// TwinCAT 3 PLC project PunchingMachine
// ProgramVersion: 3.1.4026.20
// libraries:
//   RMTH TC3 Library, * (RMTH GmbH)
//   Tc2_Drive, * (Beckhoff Automation GmbH)
//   Tc2_EtherCAT, * (Beckhoff Automation GmbH)
//   Tc2_MC2, * (Beckhoff Automation GmbH)
//   Tc2_MC2_Drive, * (Beckhoff Automation GmbH)
//   Tc2_NC, * (Beckhoff Automation GmbH)
//   Tc2_NCI, * (Beckhoff Automation GmbH)
//   Tc2_Standard, * (Beckhoff Automation GmbH)
//   Tc2_System, * (Beckhoff Automation GmbH)
//   Tc2_Utilities, * (Beckhoff Automation GmbH)
//   Tc3_EventLogger, * (Beckhoff Automation GmbH)
//   Tc3_Module, * (Beckhoff Automation GmbH)
//   BASIC,3.3.3.0,OSCAT
// project tree:
//   BaseComponents/AxisDriver/Enumeration/ E_GearMode.TcDUT, E_JogDirection.TcDUT, E_MotionCommand.TcDUT
//   BaseComponents/AxisDriver/ FB_AxisDriver.TcPOU
//   BaseComponents/AxisDriver/Interfaces/ ITFMotionComponent.TcIO
//   BaseComponents/AxisDriver/Structures/AdditionalAxisIO/ ST_AxisIn.TcDUT, ST_AxisIO.TcDUT, ST_AxisOut.TcDUT, ST_AxisVirtualIO.TcDUT
//   BaseComponents/AxisDriver/Structures/ ST_AxisDriverParameter.TcDUT, ST_AxisGearInParameter.TcDUT, ST_AxisGearOutParameter.TcDUT, ST_AxisGeneralParameter.TcDUT, ST_AxisHaltParameter.TcDUT, ST_AxisHomingParameter.TcDUT, ST_AxisJogAccParameter.TcDUT, ST_AxisJogParameter.TcDUT, ST_AxisMoveAbsParameter.TcDUT, ST_AxisMoveAddParameter.TcDUT, ST_AxisMoveModParameter.TcDUT, ST_AxisMoveParameter.TcDUT, ST_AxisMoveRelParameter.TcDUT, ST_AxisMoveVelParameter.TcDUT, ST_AxisSetPosParameter.TcDUT, ST_AxisStopParameter.TcDUT
//   BaseComponents/AxisDriver/Utilities/ FB_AxisDistanceTrigger.TcPOU, FB_LimitSwitchRefSim.TcPOU, F_LRealToString.TcPOU, F_LRealToStringEx.TcPOU, F_SpeedReached.TcPOU, F_SpeedWindowReached.TcPOU, F_TargetReached.TcPOU, F_TargetReachedOrHigher.TcPOU, F_TargetReachedOrLower.TcPOU, F_TargetWindowReached.TcPOU, F_TargetWindowReachedAxisRef.TcPOU
//   BaseComponents/CylinderDriver/Enumeration/ E_CylinderPosition.TcDUT
//   BaseComponents/CylinderDriver/ FB_CylinderDriver.TcPOU
//   BaseComponents/CylinderDriver/Interfaces/ ITF_Cylinder.TcIO
//   BaseComponents/CylinderDriver/Structures/ ST_CylinderDriverIn.TcDUT, ST_CylinderDriverIO.TcDUT, ST_CylinderDriverOut.TcDUT
//   BaseComponents/DigitalInput/ FB_DigitalInput.TcPOU
//   BaseComponents/DigitalInput/Structures/ ST_DigitalInputIn.TcDUT, ST_DigitalInputIO.TcDUT
//   BaseComponents/DigitalOutput/ FB_DigitalOutput.TcPOU
//   BaseComponents/DigitalOutput/Structures/ ST_DigitalOutputIO.TcDUT, ST_DigitalOutputOUT.TcDUT
//   BaseComponents/EtherCAT/Enumerations/ E_EtherCatSlaveState.TcDUT, E_EtherCATState.TcDUT
//   BaseComponents/EtherCAT/ FB_EtherCatBox.TcPOU, FB_EtherCATBus.TcPOU
//   BaseComponents/EtherCAT/Structures/ ST_EtherCatBoxIO.TcDUT, ST_EtherCatIO.TcDUT
//   BaseComponents/EventLog/Enumerations/ E_BoolFilter.TcDUT, E_FilterActive.TcDUT, E_Priority.TcDUT
//   BaseComponents/EventLog/ E_Event.TcDUT, FB_EventLog.TcPOU
//   BaseComponents/EventLog/Structures/ ST_Event.TcDUT, ST_EventFilter.TcDUT
//   BaseComponents/SafetyLockDriver/ FB_SafetyLock.TcPOU
//   BaseComponents/SafetyLockDriver/Structures/ ST_SafetyLockIn.TcDUT, ST_SafetyLockIO.TcDUT, ST_SafetyLockOut.TcDUT
//   BaseComponents/Safety/ FB_Safety.TcPOU
//   BaseComponents/Safety/Structures/ ST_SafetyIn.TcDUT, ST_SafetyIO.TcDUT, ST_SafetyOut.TcDUT
//   BaseComponents/Supervision/CheckFunctions/ CheckBounds.TcPOU, CheckDivDInt.TcPOU, CheckDivLInt.TcPOU, CheckDivLReal.TcPOU, CheckDivReal.TcPOU, CheckPointer.TcPOU, CheckRangeSigned.TcPOU, CheckRangeUnsigned.TcPOU
//   BaseComponents/Supervision/Enumeration/ E_CodeError.TcDUT
//   BaseComponents/Supervision/ FB_Supervision.TcPOU, GVL_Supervision.TcGVL
//   Components/ E_ComponentType.TcDUT
//   Components/MatAndToolHandling/Enumerations/ E_MatAndToolHandlingCmd.TcDUT
//   Components/MatAndToolHandling/ FB_MatAndToolHandling.TcPOU
//   Components/Mat/Enumerations/ E_CoordinatesSortState.TcTLEO, E_Geometry.TcDUT, E_ElementOrigin.TcDUT
//   Components/Mat/ FB_Mat.TcPOU
//   Components/Mat/Structures/ ST_Element.TcDUT, ST_Mat.TcDUT, ST_MatRun.TcDUT, ST_Tool.TcDUT, ST_ToolHolder.TcDUT, ST_Coordinate.TcDUT
//   Components/PunchEngine/Enumerations/ E_PunchEngineCmd.TcDUT
//   Components/PunchEngine/ FB_PunchEngine.TcPOU
//   / IOTask.TcTTO, NcTask.TcTTO, PlcTask.TcTTO, VisuTask.TcTTO
//   Machine/Components/ E_Axis.TcDUT, E_DigitalOutput.TcDUT, E_Cylinder.TcDUT, COMP_CONST.TcGVL, COMP.TcGVL
//   Machine/Enumerations/ E_JobState.TcDUT, E_MachineArea.TcDUT, E_OperationMode.TcDUT, E_RunTodo.TcDUT
//   Machine/ GVL.TcGVL, GVL_CONST.TcGVL, P_Machine.TcPOU
//   Machine/Structures/ ST_MachineConfig.TcDUT, ST_PunchJob.TcDUT
//   Utilities/Component/Enumerations/ E_ComponentState.TcDUT
//   Utilities/Component/ FB_ComponentBase.TcPOU
//   Utilities/Component/Interfaces/ ITFComponent.TcIO
//   Utilities/Composition/ FB_CompositionBase.TcPOU
//   Utilities/Sequencer/Enumeration/ E_SequenceState.TcDUT
//   Utilities/Sequencer/ FB_Sequence.TcPOU
//   Utilities/TaskAllocation/Enumerations/ E_Task.TcDUT
//   Utilities/TaskAllocation/ P_Fast.TcPOU
//   Utilities/TaskAllocation/Interfaces/ ITF_TaskAllocation.TcIO
//   Visualisation/Structures/ ST_MaintCmds.TcDUT, ST_MaintParam.TcDUT, ST_PunchCmds.TcDUT, ST_PunchInfo.TcDUT, ST_MaintInfo.TcDUT, ST_PunchParam.TcDUT
//   Visualisation/ GVL_VISU.TcGVL, P_Visu.TcPOU
// real-time tasks:
//   TASK PlcTask: cycle T#10ms, priority 14, ADS port 350
//   TASK NcTask: cycle T#10ms, priority 12, ADS port 351
//   TASK IOTask: cycle T#10ms, priority 8, ADS port 354
//   TASK VisuTask: cycle T#50000us, priority 16, ADS port 353
// motion (NC):
//   TASK NC-Task 1 SAF: cycle T#2ms, priority 4, ADS port 501
//   TASK NC-Task 1 SVB: cycle T#10ms, priority 10, ADS port 511
//   AXIS x-Axis (id 4)
//     Dynamic: Acceleration=5500, Deceleration=5500, Jerk=15000
//     Velo: RefSearch=18.6430234375, RefSync=18.6430234375, SlowManual=10, FastManual=250, Fast=1864.30234375, Maximum=1864.3
//     OtherSettings: AllowMotionCmdToSlave=true
//     encoder EncType=8
//       EncPara: ScaleFactorNumerator=41.5555555555556, ScaleFactorDenominator=1048576, Offset=17493, MaxCount=#xffffffff
//         SoftEndMinControl: Enable=true
//         SoftEndMaxControl: Enable=true, Range=4070
//     drive DrvType=9
//       DrvPara: MaxCount=#xffffffff, DriveControlDWord=#x00030100
//         Analog: VeloReferenz=2050.732578125, VeloScale=1.02400649589962, ScaleFactorActTorque=0.1
//         TimeComp: TaskDelayCycles=1
//     controller CtrType=1
//       CtrPara: PriorControlFactor=1
//         Observer: BandWidth=20
//   AXIS y-Axis (id 5)
//     Dynamic: Acceleration=11000, Deceleration=11000, Jerk=30000
//     Velo: RefSearch=32.25, RefSync=32.25, SlowManual=161.25, FastManual=967.5, Fast=3225, Maximum=3225
//     OtherSettings: AllowMotionCmdToSlave=true
//     encoder EncType=8
//       EncPara: ScaleFactorNumerator=21.5, ScaleFactorDenominator=1048576, Offset=-280, Inverse=true, MaxCount=#xffffffff
//         SoftEndMinControl: Enable=true, Range=5
//         SoftEndMaxControl: Enable=true, Range=790
//     drive DrvType=9
//       DrvPara: Inverse=true, MaxCount=#xffffffff, DriveControlDWord=#x00030100
//         Analog: VeloReferenz=3547.5, VeloScale=1.02400649589962, ScaleFactorActTorque=0.1
//         TimeComp: TaskDelayCycles=1
//     controller CtrType=1
//       CtrPara: PriorControlFactor=1
//         Observer: BandWidth=20
//   AXIS PunchAxis (id 6)
//     General: UnitName=Degree, UnitFlags=#x00000004
//     Dynamic: Acceleration=10000, Deceleration=10000, Jerk=100000
//     Velo: RefSearch=11.1429969216489, RefSync=11.1429969216489, SlowManual=55.7149846082443, FastManual=900, Fast=1114.29969216489, Maximum=1114.3
//     PositionAreaControl: Enable=false
//     TargetPosControl: Enable=false
//     OtherSettings: AllowMotionCmdToSlave=true
//     encoder EncType=8
//       EncPara: ScaleFactorNumerator=20.1237295625276, ScaleFactorDenominator=1048576, Offset=-12, ToleranceWndModuloStart=1.5, MaxCount=#x000fffff
//     drive DrvType=9
//       DrvPara: MaxCount=#xffffffff, DriveControlDWord=#x00030100
//         Analog: VeloReferenz=1225.72966138138, VeloScale=1.02400649589962, ScaleFactorActTorque=0.1
//         TimeComp: TaskDelayCycles=1
//     controller CtrType=1
//       CtrPara: PriorControlFactor=1
//         PosDiffControl: Enable=false
//         Observer: BandWidth=20
// I/O:
//   DEVICE Device 2 (EtherCAT), AmsNetId 192.168.137.129.3.1
//     Term 1 (EK1100) [EK1100 EtherCAT Coupler (2A E-Bus)]
//       Term 2 (EL6910) [EL6910, TwinSAFE PLC]
//       Term 3 (EL2904) [EL2904, 4 Ch. Safety Output 24V, 0.5A, TwinSAFE]
//         modules: Module 1 (FSOES), Module 2 (DO)
//       Term 4 (EL1904) [EL1904, 4 Ch. Safety Input 24V, TwinSAFE]
//         modules: Module 1 (FSOES)
//       Term 5 (EL1904) [EL1904, 4 Ch. Safety Input 24V, TwinSAFE]
//         modules: Module 1 (FSOES)
//       Term 6 (EL1008) [EL1008 8Ch. Dig. Input 24V, 3ms]
//       Term 7 (EL1008) [EL1008 8Ch. Dig. Input 24V, 3ms]
//       Term 8 (EL2008) [EL2008 8Ch. Dig. Output 24V, 0.5A]
//       Term 13 (EL9011) [EL9011 End Terminal]
//     Drive 9 (AX5206-0000-0210) [AX5206-0000-0210 EtherCAT Drive (SoE, 2 Ch.)]
//       Term 10 (AX5805) [AX5805 (Safety Drive Option)]
//         modules: Module 1 (Safety Process Data, 2 axis), Module 2 (Standard Process Data, 2 axis)
//       Term 14 (EL9011) [EL9011 End Terminal]
//     Drive 11 (AX5112-0000-0210) [AX5112-0000-0210 EtherCAT Drive (SoE, 1 Ch.)]
//       Term 12 (AX5805) [AX5805 (Safety Drive Option)]
//         modules: Module 1 (Safety Process Data, 1 axis), Module 2 (Standard Process Data, 1 axis)
//       Term 15 (EL9011) [EL9011 End Terminal]
// variable links:
//   Device 2 (EtherCAT) <-> Device 2 (EtherCAT)/Drive 11 (AX5112-0000-0210)/Term 12 (AX5805)
//     Term 1 (EK1100)/Term 2 (EL6910)/ConnectionInputs/Message_7 TxPDO <-> Module 1 (Safety Process Data, 1 axis)/Outputs (Controlword)/FSOE
//     Term 1 (EK1100)/Term 2 (EL6910)/ConnectionOutputs/Message_7 RxPDO <-> Module 1 (Safety Process Data, 1 axis)/Inputs (Statusword)/FSOE
//   Device 2 (EtherCAT) <-> Device 2 (EtherCAT)/Drive 9 (AX5206-0000-0210)/Term 10 (AX5805)
//     Term 1 (EK1100)/Term 2 (EL6910)/ConnectionInputs/Message_6 TxPDO <-> Module 1 (Safety Process Data, 2 axis)/Outputs (Controlword)/FSOE
//     Term 1 (EK1100)/Term 2 (EL6910)/ConnectionOutputs/Message_6 RxPDO <-> Module 1 (Safety Process Data, 2 axis)/Inputs (Statusword)/FSOE
//   Device 2 (EtherCAT) <-> Device 2 (EtherCAT)/Term 1 (EK1100)/Term 3 (EL2904)
//     Term 1 (EK1100)/Term 2 (EL6910)/ConnectionInputs/Message_16 TxPDO <-> Module 1 (FSOES)/RxPDO/FSOE
//     Term 1 (EK1100)/Term 2 (EL6910)/ConnectionOutputs/Message_16 RxPDO <-> Module 1 (FSOES)/TxPDO/FSOE
//   Device 2 (EtherCAT) <-> Device 2 (EtherCAT)/Term 1 (EK1100)/Term 4 (EL1904)
//     Term 1 (EK1100)/Term 2 (EL6910)/ConnectionInputs/Message_4 TxPDO <-> Module 1 (FSOES)/RxPDO/FSOE
//     Term 1 (EK1100)/Term 2 (EL6910)/ConnectionOutputs/Message_4 RxPDO <-> Module 1 (FSOES)/TxPDO/FSOE
//   Device 2 (EtherCAT) <-> Device 2 (EtherCAT)/Term 1 (EK1100)/Term 5 (EL1904)
//     Term 1 (EK1100)/Term 2 (EL6910)/ConnectionInputs/Message_17 TxPDO <-> Module 1 (FSOES)/RxPDO/FSOE
//     Term 1 (EK1100)/Term 2 (EL6910)/ConnectionOutputs/Message_17 RxPDO <-> Module 1 (FSOES)/TxPDO/FSOE
//   NC-Task 1 SAF/Axes/PunchAxis <-> Device 2 (EtherCAT)/Drive 11 (AX5112-0000-0210)
//     Drive/Inputs/In/nDataIn1 <-> AT/Following distance
//     Drive/Inputs/In/nDcOutputTime <-> InfoData/DcOutputShift
//     Drive/Inputs/In/nState1 <-> AT/Drive status word @bit 8
//     Drive/Inputs/In/nState2 <-> AT/Drive status word
//     Drive/Inputs/In/nState4 @bit 1 <-> WcState/InputToggle
//     Drive/Inputs/In/nState4 <-> WcState/WcState
//     Drive/Outputs/Out/nCtrl1 <-> MDT/Master control word @bit 8
//     Drive/Outputs/Out/nDataOut1 <-> MDT/Position command value
//     Enc/Inputs/In/nDataIn1 <-> AT/Position feedback 1 value
//     Enc/Inputs/In/nDcInputTime <-> InfoData/DcInputShift
//     Enc/Inputs/In/nState4 @bit 1 <-> WcState/InputToggle
//     Enc/Inputs/In/nState4 <-> WcState/WcState
//   NC-Task 1 SAF/Axes/x-Axis <-> Device 2 (EtherCAT)/Drive 9 (AX5206-0000-0210)
//     Drive/Inputs/In/nDataIn1 <-> AT 1/Following distance
//     Drive/Inputs/In/nDcOutputTime <-> InfoData/DcOutputShift
//     Drive/Inputs/In/nState1 <-> AT 1/Drive status word @bit 8
//     Drive/Inputs/In/nState2 <-> AT 1/Drive status word
//     Drive/Inputs/In/nState4 @bit 1 <-> WcState/InputToggle
//     Drive/Inputs/In/nState4 <-> WcState/WcState
//     Drive/Outputs/Out/nCtrl1 <-> MDT 1/Master control word @bit 8
//     Drive/Outputs/Out/nDataOut1 <-> MDT 1/Position command value
//     Enc/Inputs/In/nDataIn1 <-> AT 1/Position feedback 1 value (motor feedback)
//     Enc/Inputs/In/nDcInputTime <-> InfoData/DcInputShift
//     Enc/Inputs/In/nState4 @bit 1 <-> WcState/InputToggle
//     Enc/Inputs/In/nState4 <-> WcState/WcState
//   NC-Task 1 SAF/Axes/y-Axis <-> Device 2 (EtherCAT)/Drive 9 (AX5206-0000-0210)
//     Drive/Inputs/In/nDataIn1 <-> AT 2/Following distance
//     Drive/Inputs/In/nDcOutputTime <-> InfoData/DcOutputShift
//     Drive/Inputs/In/nState1 <-> AT 2/Drive status word @bit 8
//     Drive/Inputs/In/nState2 <-> AT 2/Drive status word
//     Drive/Inputs/In/nState4 @bit 1 <-> WcState/InputToggle
//     Drive/Inputs/In/nState4 <-> WcState/WcState
//     Drive/Outputs/Out/nCtrl1 <-> MDT 2/Master control word @bit 8
//     Drive/Outputs/Out/nDataOut1 <-> MDT 2/Position command value
//     Enc/Inputs/In/nDataIn1 <-> AT 2/Position feedback 1 value
//     Enc/Inputs/In/nDcInputTime <-> InfoData/DcInputShift
//     Enc/Inputs/In/nState4 @bit 1 <-> WcState/InputToggle
//     Enc/Inputs/In/nState4 <-> WcState/WcState
//   PunchingMachine/PunchingMachine Instance <-> Device 2 (EtherCAT)/Drive 11 (AX5112-0000-0210)
//     NcTask Inputs/COMP.astAxisIO[2].stIn/iAmplifierTemperature <-> AT/Heatsink temperature
//     NcTask Inputs/COMP.astAxisIO[2].stIn/iMotorTemperature <-> AT/Motor temperature
//     NcTask Inputs/COMP.astAxisIO[2].stIn/iTorqueFeedbackValue <-> AT/Torque/force feedback value
//     NcTask Outputs/COMP.astAxisIO[2].stOut/iBipolarTorqueLimitValue <-> MDT/Bipolar torque/force limit value
//     NcTask Outputs/COMP.astAxisIO[2].stOut/iNegativeTorqueLimitValue <-> MDT/Negative torque/force limit value
//     NcTask Outputs/COMP.astAxisIO[2].stOut/iPositiveTorqueLimitValue <-> MDT/Positive torque/force limit value
//   PunchingMachine/PunchingMachine Instance <-> Device 2 (EtherCAT)/Drive 9 (AX5206-0000-0210)
//     NcTask Inputs/COMP.astAxisIO[0].stIn/iAmplifierTemperature <-> AT 1/Heatsink temperature
//     NcTask Inputs/COMP.astAxisIO[1].stIn/iAmplifierTemperature <-> AT 2/Heatsink temperature
//     NcTask Inputs/COMP.astAxisIO[0].stIn/iMotorTemperature <-> AT 1/Motor temperature
//     NcTask Inputs/COMP.astAxisIO[1].stIn/iMotorTemperature <-> AT 2/Motor temperature
//     NcTask Inputs/COMP.astAxisIO[0].stIn/iTorqueFeedbackValue <-> AT 1/Torque/force feedback value
//     NcTask Inputs/COMP.astAxisIO[1].stIn/iTorqueFeedbackValue <-> AT 2/Torque/force feedback value
//     NcTask Outputs/COMP.astAxisIO[0].stOut/iBipolarTorqueLimitValue <-> MDT 1/Bipolar torque/force limit value
//     NcTask Outputs/COMP.astAxisIO[1].stOut/iBipolarTorqueLimitValue <-> MDT 2/Bipolar torque/force limit value
//     NcTask Outputs/COMP.astAxisIO[0].stOut/iNegativeTorqueLimitValue <-> MDT 1/Negative torque/force limit value
//     NcTask Outputs/COMP.astAxisIO[1].stOut/iNegativeTorqueLimitValue <-> MDT 2/Negative torque/force limit value
//     NcTask Outputs/COMP.astAxisIO[0].stOut/iPositiveTorqueLimitValue <-> MDT 1/Positive torque/force limit value
//     NcTask Outputs/COMP.astAxisIO[1].stOut/iPositiveTorqueLimitValue <-> MDT 2/Positive torque/force limit value
//   PunchingMachine/PunchingMachine Instance <-> Device 2 (EtherCAT)/Term 1 (EK1100)/Term 2 (EL6910)
//     IOTask Inputs/COMP.stSafetyIO.stIn.bSAFE_CommErr <-> StandardInputs/Standard Out Var 11
//     IOTask Inputs/COMP.stSafetyIO.stIn.bSAFE_FbErr <-> StandardInputs/Standard Out Var 12
//     IOTask Inputs/COMP.stSafetyIO.stIn.bSAFE_NotHalt_Ok <-> StandardInputs/Standard Out Var 9
//     IOTask Inputs/COMP.stSafetyLockIO.stIn.bSaftyOK <-> StandardInputs/Standard Out Var 18
//     IOTask Outputs/COMP.stSafetyIO.stOut/bErrAckSafety_Drive <-> StandardOutputs/Standard In Var 10
//     IOTask Outputs/COMP.stSafetyIO.stOut/bErrAckSafety_General <-> StandardOutputs/Standard In Var 1
//     IOTask Outputs/COMP.stSafetyIO.stOut/bRun_stop <-> StandardOutputs/Standard In Var 14
//   PunchingMachine/PunchingMachine Instance <-> Device 2 (EtherCAT)/Term 1 (EK1100)/Term 3 (EL2904)
//     IOTask Outputs/COMP.aStCylinderIO[0].stOut/bValveCylinderHp <-> Module 2 (DO)/RxPDO/bValveCylinderHp
//     IOTask Outputs/COMP.aStCylinderIO[0].stOut/bValveCylinderWp <-> Module 2 (DO)/RxPDO/bValveCylinderWp
//     IOTask Outputs/COMP.stSafetyIO.stOut/bSAFE_NotHalt_Ok <-> Module 2 (DO)/RxPDO/Output Channel 1
//     IOTask Outputs/COMP.stSafetyIO.stOut/bSAFE_NotHalt_Ok <-> Module 2 (DO)/RxPDO/Output Channel 2
//   PunchingMachine/PunchingMachine Instance <-> Device 2 (EtherCAT)/Term 1 (EK1100)/Term 7 (EL1008)
//     IOTask Inputs/COMP.aStCylinderIO[0].stIn/bCylinderSensorHp <-> Channel 8/bCylinderSensorHp
//     IOTask Inputs/COMP.aStCylinderIO[0].stIn/bCylinderSensorWp <-> Channel 7/bCylinderSensorWp
//   PunchingMachine/PunchingMachine Instance <-> Device 2 (EtherCAT)/Term 1 (EK1100)/Term 8 (EL2008)
//     IOTask Outputs/COMP.aStDigitalOutputIO[0].stOut/bOutput <-> Channel 2/bOutput
//     IOTask Outputs/COMP.stSafetyLockIO.stOut/bLock <-> Channel 1/Output
//   PunchingMachine/PunchingMachine Instance <-> NC-Task 1 SAF/Axes/PunchAxis
//     NcTask Inputs/COMP.astAxisRef[2].NcToPlc <-> Outputs/ToPlc
//     NcTask Outputs/COMP.astAxisRef[2].PlcToNc <-> Inputs/FromPlc
//   PunchingMachine/PunchingMachine Instance <-> NC-Task 1 SAF/Axes/x-Axis
//     NcTask Inputs/COMP.astAxisRef[0].NcToPlc <-> Outputs/ToPlc
//     NcTask Outputs/COMP.astAxisRef[0].PlcToNc <-> Inputs/FromPlc
//   PunchingMachine/PunchingMachine Instance <-> NC-Task 1 SAF/Axes/y-Axis
//     NcTask Inputs/COMP.astAxisRef[1].NcToPlc <-> Outputs/ToPlc
//     NcTask Outputs/COMP.astAxisRef[1].PlcToNc <-> Inputs/FromPlc

CONFIGURATION PunchingMachine
    RESOURCE PLC ON TwinCAT3
        TASK IOTask(INTERVAL := T#10ms, PRIORITY := 8);
        TASK NcTask(INTERVAL := T#10ms, PRIORITY := 12);
        TASK PlcTask(INTERVAL := T#10ms, PRIORITY := 14);
        TASK VisuTask(INTERVAL := T#50000us, PRIORITY := 16);
        PROGRAM P_Machine WITH PlcTask : P_Machine;
        PROGRAM P_System WITH PlcTask : P_System;
        PROGRAM P_Visu WITH VisuTask : P_Visu;
    END_RESOURCE
END_CONFIGURATION

// ---- BaseComponents/AxisDriver/Enumeration/E_GearMode.TcDUT
/// Enumeration of possible axis gear modes.
TYPE E_GearMode :
(
	/// Gear mode not set
	eGearMode_none := 0,
	/// Gear in
	eGearMode_in,
	/// Gear out
	eGearMode_out
);
END_TYPE

// ---- BaseComponents/AxisDriver/Enumeration/E_JogDirection.TcDUT
/// Enumeration of possible jog directions.
TYPE E_JogDirection :
(
	/// Jog direction not set
	eJogDirection_none := 0,
	/// Jog direction positive
	eJogDirection_pos,
	/// Jog direction negative
	eJogDirection_neg
);
END_TYPE

// ---- BaseComponents/AxisDriver/Enumeration/E_MotionCommand.TcDUT
/// Enumeration of possible axis motion commands.
TYPE E_MotionCommand :
(
	/// No command
	eMotionCommand_none := 0,
	/// Reset axis
	eMotionCommand_reset := 1,
	/// Axis halt (default stopping method)
	eMotionCommand_halt := 2,
	/// Axis stop (needs reset before next motion command)
	eMotionCommand_stop := 3,
	/// Axis homing
	eMotionCommand_home := 4,
	/// Set axis position
	eMotionCommand_setPos := 5,
	/// Jog axis
	eMotionCommand_jog := 6,
	/// Jog axis accelerating
	eMotionCommand_jogAcc := 7,
	/// Move axis to point
	eMotionCommand_moveAbs := 8,
	/// Move axis additive
	eMotionCommand_moveAdd := 9,
	/// Move axis relative
	eMotionCommand_moveRel := 10,
	/// Move axis modulo
	eMotionCommand_moveMod := 11,
	/// Move axis velocity (endles)
	eMotionCommand_moveVel := 12,
	/// Apply axis torque
	eMotionCommand_torque := 13,
	/// Gear axis in (electronic) or change gear ratio
	eMotionCommand_gearIn := 14,
	/// Gear axis out (electronic), default behavior: halt axis after gear out
	eMotionCommand_gearOut := 15,
	/// Axis start/stop touch probe
	eMotionCommand_touchProbe := 16,
	/// Set override in maintenance mode
	eMotionCommand_setOverride := 17
);
END_TYPE

// ---- BaseComponents/AxisDriver/Structures/AdditionalAxisIO/ST_AxisIn.TcDUT
TYPE ST_AxisIn :
STRUCT
	/// Torque from drive [1/10 Nm]
	iTorqueFeedbackValue	: INT;
	/// Motortemp: [1/10 °C]
	iMotorTemperature		: INT;
	/// Amplifiertemp: [1/10 °C]
	iAmplifierTemperature	: INT;
	/// calibration Sensor
	bCalibrationCam			: BOOL;
	/// Limit Sensor Pos
	bLimitPos				: BOOL;
	/// Limit Sensor Neg
	bLimitNeg				: BOOL;
	/// Limit Sensor Neg
	nPositionFeedbackValue	: DINT;
END_STRUCT
END_TYPE

// ---- BaseComponents/AxisDriver/Structures/AdditionalAxisIO/ST_AxisIO.TcDUT
/// Additional axis IO (direct linked) for AX5xxx axis.
TYPE ST_AxisIO :
STRUCT
	stIn AT %I*: ST_AxisIn;
	stOut AT %Q*: ST_AxisOut;
END_STRUCT
END_TYPE

// ---- BaseComponents/AxisDriver/Structures/AdditionalAxisIO/ST_AxisOut.TcDUT
TYPE ST_AxisOut :
STRUCT
	/// Ext. fan control
	bExternalFan: BOOL;
	/// The bipolar torque limit value limits the maximum torque symmetrically in both directions. [1/10 %]
	iBipolarTorqueLimitValue: INT := 1000;
	iPositiveTorqueLimitValue: INT := 1000;
	iNegativeTorqueLimitValue: INT := 1000;
END_STRUCT
END_TYPE

// ---- BaseComponents/AxisDriver/Structures/AdditionalAxisIO/ST_AxisVirtualIO.TcDUT
/// Dummy IO for virtual axis.
TYPE ST_AxisVirtualIO :
STRUCT
	stIn: ST_AxisIn;
	stOut: ST_AxisOut;
END_STRUCT
END_TYPE

// ---- BaseComponents/AxisDriver/Structures/ST_AxisDriverParameter.TcDUT
/// Parameter set for axis driver
TYPE ST_AxisDriverParameter :
STRUCT
	/// General axis parameter
	stGeneralPrm: ST_AxisGeneralParameter;
	/// Parameter for halting the axis
	stHaltPrm: ST_AxisHaltParameter;
	/// Parameter for stopping the axis
	stStopPrm: ST_AxisStopParameter;
	/// Parameter for axis homing
	stHomingPrm: ST_AxisHomingParameter;
	/// Parameter for axis set position
	stSetPosPrm: ST_AxisSetPosParameter;
	/// Parameter for axis homing
	stJogPrm: ST_AxisJogParameter;
	/// Parameter for accelerating jog
	stJogAccPrm: ST_AxisJogAccParameter;
	/// Parameter for move axis absolute
	stMovAbsPrm: ST_AxisMoveAbsParameter;
	/// Parameter for move axis additive
	stMovAddPrm: ST_AxisMoveAddParameter;
	/// Parameter for move axis relative
	stMovRelPrm: ST_AxisMoveRelParameter;
	/// Parameter for move axis modulo
	stMovModPrm: ST_AxisMoveModParameter;
	/// Parameter for move axis velocity
	stMovVelPrm: ST_AxisMoveVelParameter;
	/// Parameter for axis electronic gear-in
	stGearInPrm: ST_AxisGearInParameter;
	/// Parameter for axis electronic gear-out
	stGearOutPrm: ST_AxisGearOutParameter;
END_STRUCT
END_TYPE

// ---- BaseComponents/AxisDriver/Structures/ST_AxisGearInParameter.TcDUT
/// GearIn parameter strucure
TYPE ST_AxisGearInParameter :
STRUCT
	eMasterId: E_Axis;
	fbMaster: REFERENCE TO AXIS_REF;
	fGearRatio: LREAL;
	fAcceleration: LREAL;
	fDeceleration: LREAL;
	fJerk: LREAL;
	eBufferMode: MC_BufferMode;
	stOptions: ST_GearInDynOptions;
END_STRUCT
END_TYPE

// ---- BaseComponents/AxisDriver/Structures/ST_AxisGearOutParameter.TcDUT
/// GearOut parameter strucure
TYPE ST_AxisGearOutParameter :
STRUCT
	/// Halt axis after gear out
	bHaltAxis: BOOL := TRUE;
	/// Gear out (not implemented)
	stOptions: ST_GearOutOptions;
END_STRUCT
END_TYPE

// ---- BaseComponents/AxisDriver/Structures/ST_AxisGeneralParameter.TcDUT
/// General axis parameter set
TYPE ST_AxisGeneralParameter :
STRUCT
	/// Auto power off axis (economize)
	bEnableAutoPowerOff: BOOL := FALSE;
	/// Delay time until power off idle axis
	tAutoPowerOffDelay: TIME := TIME#10s0ms;
	/// Threshold temperature [1/10 °C] for external fan.
	iExtFanThreshold: INT := 500;
	/// Factor for torque value
	fTorqueFactor: REAL := 0.1;
END_STRUCT
END_TYPE

// ---- BaseComponents/AxisDriver/Structures/ST_AxisHaltParameter.TcDUT
TYPE ST_AxisHaltParameter EXTENDS ST_AxisStopParameter :
STRUCT
	eBufferMode: MC_BufferMode := MC_Aborting;
END_STRUCT
END_TYPE

// ---- BaseComponents/AxisDriver/Structures/ST_AxisHomingParameter.TcDUT
TYPE ST_AxisHomingParameter :
STRUCT
	bCalibrationCam: REFERENCE TO BOOL;
	fPosition: LREAL := DEFAULT_HOME_POSITION;
	eHomingMode: MC_HomingMode := MC_DefaultHoming;
	eBufferMode: MC_BufferMode := MC_Aborting;
	stOptions: ST_HomingOptions;
END_STRUCT
END_TYPE

// ---- BaseComponents/AxisDriver/Structures/ST_AxisJogAccParameter.TcDUT
/// Accelerating jog parameter strucure
TYPE ST_AxisJogAccParameter EXTENDS ST_AxisMoveParameter :
STRUCT
	/// Jog axis backward
	bJogBackwards: BOOL;
	/// Jog axis forward
	bJogForward: BOOL;
	/// Slow (starting) speed
	fSlowSpeed: LREAL;
	/// Fast end-speed
	fFastSpeed: LREAL;
	/// Time for ramp from slow to fast speed 
	tAccTime: TIME;
END_STRUCT
END_TYPE

// ---- BaseComponents/AxisDriver/Structures/ST_AxisJogParameter.TcDUT
/// Axis jog parameter strucure
TYPE ST_AxisJogParameter :
STRUCT
	bJogBackwards: BOOL;
	bJogForward: BOOL;
	fAcceleration: LREAL;
	fDeceleration: LREAL;
	fJerk: LREAL;
	eMode: E_JogMode;
	fPosition: LREAL;
	fVelocity: LREAL;
END_STRUCT
END_TYPE

// ---- BaseComponents/AxisDriver/Structures/ST_AxisMoveAbsParameter.TcDUT
/// Axis move absolute parameter strucure
TYPE ST_AxisMoveAbsParameter EXTENDS ST_AxisMoveParameter :
STRUCT
	fPosition: LREAL;
END_STRUCT
END_TYPE

// ---- BaseComponents/AxisDriver/Structures/ST_AxisMoveAddParameter.TcDUT
/// Axis move additive parameter strucure
TYPE ST_AxisMoveAddParameter EXTENDS ST_AxisMoveParameter :
STRUCT
	/// Distance
	fDistance: LREAL;
END_STRUCT
END_TYPE

// ---- BaseComponents/AxisDriver/Structures/ST_AxisMoveModParameter.TcDUT
/// Axis move modulo parameter strucure
TYPE ST_AxisMoveModParameter EXTENDS ST_AxisMoveParameter :
STRUCT
	fPosition: LREAL;
	eDirection: MC_Direction;
END_STRUCT
END_TYPE

// ---- BaseComponents/AxisDriver/Structures/ST_AxisMoveParameter.TcDUT
/// General move parameter strucure
TYPE ST_AxisMoveParameter :
STRUCT
	fVelocity: LREAL;
	fAcceleration: LREAL;
	fDeceleration: LREAL;
	fJerk: LREAL;
	eBufferMode: MC_BufferMode := MC_Aborting;
	stOptions: ST_MoveOptions;
END_STRUCT
END_TYPE

// ---- BaseComponents/AxisDriver/Structures/ST_AxisMoveRelParameter.TcDUT
/// Axis move relative parameter strucure
TYPE ST_AxisMoveRelParameter EXTENDS ST_AxisMoveParameter :
STRUCT
	/// Distance
	fDistance: LREAL;
END_STRUCT
END_TYPE

// ---- BaseComponents/AxisDriver/Structures/ST_AxisMoveVelParameter.TcDUT
/// Axis move velocity parameter strucure
TYPE ST_AxisMoveVelParameter EXTENDS ST_AxisMoveParameter :
STRUCT
	eDirection: MC_Direction;
END_STRUCT
END_TYPE

// ---- BaseComponents/AxisDriver/Structures/ST_AxisSetPosParameter.TcDUT
/// Parameter set for set axis position
TYPE ST_AxisSetPosParameter :
STRUCT
	/// Position to set
	fPosition: LREAL;
	/// RELATIVE=True, ABSOLUTE=False (Default)
	bMode: BOOL;
	/// Additional set position options
	stOptions: ST_SetPositionOptions;
END_STRUCT
END_TYPE

// ---- BaseComponents/AxisDriver/Structures/ST_AxisStopParameter.TcDUT
TYPE ST_AxisStopParameter :
STRUCT
	fDeceleration: LREAL;
	fJerk: LREAL;
	stOptions: ST_MoveOptions;
END_STRUCT
END_TYPE

// ---- BaseComponents/CylinderDriver/Enumeration/E_CylinderPosition.TcDUT
TYPE E_CylinderPosition :
(
	eCylinderPosition_unknown := 0,
	eCylinderPosition_hp,
	eCylinderPosition_mp,
	eCylinderPosition_wp
);
END_TYPE

// ---- BaseComponents/CylinderDriver/Structures/ST_CylinderDriverIn.TcDUT
TYPE ST_CylinderDriverIn :
STRUCT
	bCylinderSensorHp	: BOOL;
	bCylinderSensorWp	: BOOL;
END_STRUCT
END_TYPE

// ---- BaseComponents/CylinderDriver/Structures/ST_CylinderDriverIO.TcDUT
TYPE ST_CylinderDriverIO :
STRUCT
	stIn 	AT%I* : ST_CylinderDriverIn;
	stOut	AT%Q* : ST_CylinderDriverOut;
END_STRUCT
END_TYPE

// ---- BaseComponents/CylinderDriver/Structures/ST_CylinderDriverOut.TcDUT
TYPE ST_CylinderDriverOut :
STRUCT
	bValveCylinderHp	: BOOL;
	bValveCylinderWp	: BOOL;
END_STRUCT
END_TYPE

// ---- BaseComponents/DigitalInput/Structures/ST_DigitalInputIn.TcDUT
TYPE ST_DigitalInputIn :
STRUCT
	bSensor		: BOOL;
END_STRUCT
END_TYPE

// ---- BaseComponents/DigitalInput/Structures/ST_DigitalInputIO.TcDUT
TYPE ST_DigitalInputIO :
STRUCT
	stIn 	AT%I* : ST_DigitalInputIn;
END_STRUCT
END_TYPE

// ---- BaseComponents/DigitalOutput/Structures/ST_DigitalOutputIO.TcDUT
TYPE ST_DigitalOutputIO :
STRUCT
	stOut 	AT%Q* : ST_DigitalOutputOut;
END_STRUCT
END_TYPE

// ---- BaseComponents/DigitalOutput/Structures/ST_DigitalOutputOUT.TcDUT
TYPE ST_DigitalOutputOUT :
STRUCT
	bOutput			: BOOL;
END_STRUCT
END_TYPE

// ---- BaseComponents/EtherCAT/Enumerations/E_EtherCatSlaveState.TcDUT
/// Listing of possible ethercat slave states
TYPE E_EtherCatSlaveState :
(
	// 0x___1 = Slave in 'INIT' state
	eEtherCatSlaveState_INIT := 0,
	// 0x___2 = Slave in 'PREOP' state
	eEtherCatSlaveState_PREOP,
	// 0x___3 = Slave in 'BOOT' state
	eEtherCatSlaveState_BOOT,
	// 0x___4 = Slave in 'SAFEOP' state
	eEtherCatSlaveState_SAFEOP,
	// 0x___8 = Slave in 'OP' state
	eEtherCatSlaveState_OP,
	// 0x001_ = Slave signals error
	eEtherCatSlaveState_SignalsError,
	// 0x002_ = Invalid vendorId, productCode... read
	eEtherCatSlaveState_Invalid,
	// 0x004_ = Initialization error occurred
	eEtherCatSlaveState_InitErr,
	// 0x008_ = Slave disabled
	eEtherCatSlaveState_Disabled,
	// 0x010_ = Slave not present
	eEtherCatSlaveState_NotPresent,
	// 0x020_ = Slave signals link error
	eEtherCatSlaveState_LinkErr,
	// 0x040_ = Slave signals missing link
	eEtherCatSlaveState_MissingLink,
	// 0x080_ = Slave signals unexpected link
	eEtherCatSlaveState_UnexpectedLink,
	// 0x100_ = Communication port A
	eEtherCatSlaveState_ComPortA,
	// 0x200_ = Communication port B
	eEtherCatSlaveState_ComPortB,
	// 0x400_ = Communication port C
	eEtherCatSlaveState_ComPortC,
	// 0x800_ = Communication port D
	eEtherCatSlaveState_ComPortD	
);
END_TYPE

// ---- BaseComponents/EtherCAT/Enumerations/E_EtherCATState.TcDUT
/// Enumeration of possible EtherCAT states.
TYPE E_EtherCATState :
(
	/// Link error
	eEtherCATState_LinkError := 1,
	/// I/O locked after link error (I/O reset required)
	eEtherCATState_IoLockedAfterLinkErr := 2,
	/// Link error (redundancy adapter)
	eEtherCATState_LinkErrRedAdapter := 4,
	/// Missing one frame (redundancy mode)
	eEtherCATState_MissingFrame := 8,
	/// Out of send resources (I/O reset required)
	eEtherCATState_OutOfSendResources := 10,
	/// Watchdog triggered
	eEtherCATState_WatchdogTriggered := 20,
	/// Ethernet driver (miniport) not found
	eEtherCATState_EthernetDrvNotFound := 40,
	/// I/O reset active
	eEtherCATState_IO_resetActive := 80,
	/// At least one device in 'INIT' state
	eEtherCATState_AtLeastOneDeviceInit := 100,
	///  At least one device in 'PRE-OP' state
	eEtherCATState_AtLeastOneDevicePreOp := 200,
	/// At least one device in 'SAFE-OP' state
	eEtherCATState_AtLeastOneDeviceSafeOp := 400,
	/// At least one device indicates an error state
	eEtherCATState_AtLeastOneDeviceError := 800,
	/// DC not in sync
	eEtherCATState_DC_notInSync := 1000
);
END_TYPE

// ---- BaseComponents/EtherCAT/Structures/ST_EtherCatBoxIO.TcDUT
/// EtherCAT IO structure
TYPE ST_EtherCatBoxIO :
STRUCT
	
	/// Data from device.
	aeEtherCatBoxState 		AT %I*	 : E_EtherCatSlaveState;	
	
	/// Data to device.           
	
END_STRUCT
END_TYPE

// ---- BaseComponents/EtherCAT/Structures/ST_EtherCatIO.TcDUT
/// EtherCAT IO structure
TYPE ST_EtherCatIO :
STRUCT
	
	/// Data from device.
	eEtherCATState			AT %I*	: 	E_EtherCATState;
	
	/// Data to device.           
	
END_STRUCT
END_TYPE

// ---- BaseComponents/EventLog/Enumerations/E_BoolFilter.TcDUT
/// Listing of possible filter to a boolean variable
TYPE E_BoolFilter :
(
	eBoolFilter_none := 0,
	eBoolFilter_true,
	eBoolFilter_false
);
END_TYPE

// ---- BaseComponents/EventLog/Enumerations/E_FilterActive.TcDUT
/// enumeration of all possible priority
TYPE E_FilterActive :
(
	eFilter_none := 0,
	eFilter_activ := 1
);
END_TYPE

// ---- BaseComponents/EventLog/Enumerations/E_Priority.TcDUT
/// enumeration of all possible priority
TYPE E_Priority :
(
	/// no priority
	ePriority_none := 0,
	/// info priority
	ePriority_info := 1,
	/// warn priority
	ePriority_warning := 2,
	/// error priority -> Zyklusstop
	ePriority_fault := 3,
	/// error priority with fast stop -> Stopp im aktuellen Schritt 
	ePriority_faultFastStop := 4,
	/// error priority with emergency stop -> Sofortstop aller Objekte
	ePriority_faultEmergency := 5
);
END_TYPE

// ---- BaseComponents/EventLog/E_Event.TcDUT
/// enumeration of all possible notifications
TYPE E_Event :
(
	/// notification not set
	eEvent_none := 0,
	/// - code errors -
	/// code error (e.g.: check bounds, check div, ...) -> additional info (error details/index/location) in dynamic content var
	eEvent_codeError := 1,
	/// - system errors -
	/// system error (e.g.: (re)started, cycletime exceeded, ...) -> additional info (index/location) in dynamic content var
	eEvent_systemError := 2,
	/// - HW errors -
	/// hardware error -> additional info (error details/index/location) in dynamic content var
	eEvent_hardwareError := 3,
	/// hardware warning -> additional info (error details/index/location) in dynamic content var
	eEvent_hardwareWarning := 4,
	/// EtherCAT Master Fehler
	eEvent_EcMasterError := 5,
	/// EtherCAT Slave Fehler
	eEvent_EcSlaveError := 6,

	// - Safety system errors -
	/// safety error -> additional info (error details/index/location) in dynamic content var
	eEvent_safetyError := 7,
	
	// - Unit Test Meldungen
	v_unitTest := 8,
	
	// bis 09
	
	// Cabinet errors
	/// Feld01 - xxx
	eEvent_Cabinet01 := 10,
	/// Feld02 - xxx
	eEvent_Cabinet02 := 11,
	/// Feld03 - xxx
	eEvent_Cabinet03 := 12,
	
	
	
	// bis 40
	
	// 40 -> Transfer System
	eEvent_transferSystemError := 40,
	
	// 50 -> Safety Fehler Schutztüre, Not-Halt, ...
	eEvent_safetyNotHalt := 50,
	eEvent_safetyArea_Machine := 51,
	eEvent_safetyArea_Robo1 := 52,
	eEvent_safetyArea_SAA := 53,
	eEvent_safetyArea_Robo2 := 54,
	eEvent_safetyArea_PA := 55,
	
	// bis 70
	
	/// Allgemein
	eEvent_generalInf := 100,
	eEvent_generalWarn := 101,
	eEvent_generalErr := 102,
	
	/// Processmodule 
	eEvent_handPmInf := 107, 
	eEvent_handPmWarn := 108, 
	eEvent_handPmErr := 109,
	
	eEvent_bestueckungPmInf := 110,
	eEvent_bestueckungPmWarn := 111,
	eEvent_bestueckungPmErr := 112,
	
	eEvent_laserPmInf := 113,
	eEvent_laserPmWarn := 114,
	eEvent_laserPmErr := 115,
	
	eEvent_kleberPmInf := 116,
	eEvent_kleberPmWarn := 117,
	eEvent_kleberPmErr := 118,
	
	eEvent_haftvermittlerPmInf := 119,
	eEvent_haftvermittlerPmWarn := 120,
	eEvent_haftvermittlerPmErr := 121,
	
	// 02 - xx
	eEvent_Lifting_01 := 200,
	eEvent_Telescop_01 := 201,
	eEvent_02_x01_Transf_fbZylGrf := 202,
	eEvent_02_x01_Station := 203,
		
	
	eEvent_InvalidCmd := 999,
	
	/// has to be set to last index for array bounds!
	eEvent_Max := 1000
);
END_TYPE

// ---- BaseComponents/EventLog/Structures/ST_Event.TcDUT
/// Event structure
TYPE ST_Event :
STRUCT
	/// INDEX in global event-Array
	nIdx				: INT;
	/// priority of the event
	ePriority			: E_Priority;
	/// ident code of the component
	nComponentID		: INT;
	/// ident code of the event
	eEventID			: E_Event;
	/// signalize
	bSignalize			: BOOL;
	/// machine area information
	eMachineArea		: E_MachineArea;
	/// Component information
	eComponent			: E_ComponentType;
	/// dynamic content info string
	sDescription		: T_MaxString;
	/// is active flag of the notification
	bIsRaised			: BOOL;
	/// raise timestamp of the notification
	dtRaiseTime			: DT;
	/// quit timestamp of the notification
	dtQuitTime			: DT;	
	/// raise timestamp of the notification in string format
	sRaiseTime			: STRING(22);
	/// quit timestamp of the notification in string format
	sQuitTime			: STRING(22);
END_STRUCT
END_TYPE

// ---- BaseComponents/EventLog/Structures/ST_EventFilter.TcDUT
/// Notification filter set
TYPE ST_EventFilter :
STRUCT
	/// Filter to IsRaised flag
	eIsRaisedFilter : E_BoolFilter := E_BoolFilter.eBoolFilter_none;
	/// Filter to priority
	ePriorityFilter	: E_Priority := E_Priority.ePriority_none;
	/// Filter to machine area
	eAreaFilter 	: E_MachineArea := E_MachineArea.eMachineArea_none;
	/// Filter Info
	eInfoFilter		: BOOL;
	/// Filter Warning
	eWarningFilter	: BOOL;
	/// Filter Info
	eErrorFilter	: BOOL;
	/// Dialog visible
	bVisible		: BOOL;
	// Default machinearea
	eDefaultMachineArea		: E_MachineArea;
END_STRUCT
END_TYPE

// ---- BaseComponents/SafetyLockDriver/Structures/ST_SafetyLockIn.TcDUT
{attribute 'pack_mode' := '0'}
TYPE ST_SafetyLockIn :
STRUCT	
	bSaftyOK		AT%I*	: BOOL;
	bButton			AT%I*	: BOOL;
END_STRUCT
END_TYPE

// ---- BaseComponents/SafetyLockDriver/Structures/ST_SafetyLockIO.TcDUT
/// Saftey Lock IO structure.
TYPE ST_SafetyLockIO :
STRUCT
	
	/// Data to device.           
	stOut		AT%Q*		: ST_SafetyLockOut;
	
	/// Data from device.
	stIn					: ST_SafetyLockIn;
	
END_STRUCT
END_TYPE

// ---- BaseComponents/SafetyLockDriver/Structures/ST_SafetyLockOut.TcDUT
{attribute 'pack_mode' := '0'}
TYPE ST_SafetyLockOut :
STRUCT
	bSaftyOk		: BOOL;
	bLock			: BOOL;
END_STRUCT
END_TYPE

// ---- BaseComponents/Safety/Structures/ST_SafetyIn.TcDUT
/// Sicherheitssignale
TYPE ST_SafetyIn :
STRUCT
	/// Not-Halt Status von Safety
	bSAFE_NotHalt_Ok						AT %I*: BOOL;
	bSAFE_CommErr							AT %I*: BOOL;
	bSAFE_FbErr								AT %I*: BOOL;
	
END_STRUCT
END_TYPE

// ---- BaseComponents/Safety/Structures/ST_SafetyIO.TcDUT
/// Safety IO's for PLC <-> TwinSAFE communication.
TYPE ST_SafetyIO :
STRUCT
	/// From TwinSAFE to PLC structure.
	stIn 					: ST_SafetyIn;
	
	/// To TwinSAFE from PLC structure.
	stOut 		AT %Q*		: ST_SafetyOut;
END_STRUCT
END_TYPE

// ---- BaseComponents/Safety/Structures/ST_SafetyOut.TcDUT
TYPE ST_SafetyOut :
STRUCT
	bSAFE_NotHalt_Ok			: BOOL;
	bErrAckSafety_General		: BOOL;
	bErrAckSafety_Drive			: BOOL;
	bRun_stop					: BOOL;
END_STRUCT
END_TYPE

// ---- BaseComponents/Supervision/Enumeration/E_CodeError.TcDUT
TYPE E_CodeError :
(
	eCodeError_none := 0,
	eCodeError_bounds := 1,
	eCodeError_divDInt := 2,
	eCodeError_divLInt := 3,
	eCodeError_divLReal := 4,
	eCodeError_divReal := 5,
	eCodeError_pointer := 6,
	eCodeError_rangeSigned := 7,
	eCodeError_rangeUnsigned := 8,
	eCodeError_maxIdx := 9
);
END_TYPE

// ---- Components/E_ComponentType.TcDUT
TYPE E_ComponentType :
(
	// BASE COMPONENTS
	eComponentType_none := 0,
	eComponentType_EtherCAT := 1,
	eComponentType_EtherCATBox := 2,
	eComponentType_Supervision := 3,	
	eComponentType_Safety := 4,	
	eComponentType_EventLog := 5,
	eComponentType_DigitalSensor := 6,
	eComponentType_DigitalOutput := 7,
	eComponentType_Axis := 8,
	eComponentType_Cylinder := 9,
	eComponentType_SafetyLock := 10,
	
	// SPECIFIC COMPONENTS
	eComponentType_PunchEngine := 100,
	eComponentType_MatAndToolHandling := 101,
	eComponentType_Mat := 102

);
END_TYPE

// ---- Components/MatAndToolHandling/Enumerations/E_MatAndToolHandlingCmd.TcDUT
{attribute 'qualified_only'}
{attribute 'strict'}
TYPE E_MatAndToolHandlingCmd :
(
	cmdNone 		:= 0,
	cmdMoveAbs 		:= 1,
	cmdHalt 		:= 2,
	cmdJog      	:= 3,
	cmdHomeing  	:= 4,
	cmdChangeTool   := 5
);
END_TYPE

// ---- Components/Mat/Enumerations/E_CoordinatesSortState.TcTLEO
{attribute 'qualified_only'}
{attribute 'strict'}
TYPE E_CoordinatesSortState :
(
	eCoordinatesSortState_undefined := 0,
	eCoordinatesSortState_unsorted := 1,
	eCoordinatesSortState_sorted := 2,
	eCoordinatesSortState_resorted_v1 := 3
);
END_TYPE

// ---- Components/Mat/Enumerations/E_Geometry.TcDUT
{attribute 'qualified_only'}
TYPE E_Geometry :
(
	eGeometry_undefined := 0,
	eGeometry_square := 1,
	eGeometry_rectangular := 2,
	eGeometry_circle := 3,
	eGeometry_point := 4
);
END_TYPE

// ---- Components/Mat/Enumerations/E_ElementOrigin.TcDUT
{attribute 'qualified_only'}
TYPE E_ElementOrigin :
(
	eElementOrigin_ButtomRight := 0,
	eElementOrigin_ButtomLeft := 1,
	eElementOrigin_TopRight := 2,
	eElementOrigin_TopLeft:= 3
);
END_TYPE

// ---- Components/Mat/Structures/ST_Element.TcDUT
TYPE ST_Element :
STRUCT
	bActive				: BOOL;
	
	fX_Pos				: REAL;
	fY_Pos				: REAL;
	
	bCentering			: BOOL;
	bMirroring			: BOOL;
	
	eOrigin				: E_ElementOrigin;
	
	nCountX				: UINT;
	fDistanceX			: REAL;
		
	nCountY				: UINT;
	fDistanceY			: REAL;
END_STRUCT
END_TYPE

// ---- Components/Mat/Structures/ST_Mat.TcDUT
TYPE ST_Mat :
STRUCT
	// Info
	nMatNr						: UINT;
	sMatName					: STRING;	
	sNotice						: STRING;
	sProductNumber				: STRING;
	                    		
	// Geometry         		
	fWidth						: REAL;
	fHeight						: REAL;
	fLenght						: REAL;
		
	astMatOrigins				: ARRAY[0..MATS_COUNT] OF ST_Coordinate;
	
	// Runs             	
	nActiveRuns					: INT;
	astRuns						: ARRAY[0..MATRUNS_COUNT] OF ST_MatRun;

END_STRUCT
END_TYPE

// ---- Components/Mat/Structures/ST_MatRun.TcDUT
TYPE ST_MatRun :
STRUCT
	bActive						: BOOL;
	// Info
	sMatRunNr					: UINT;	
	sMatRunName					: STRING;
	sNotice						: T_MAXSTRING;

	// Punching Parameters
	fMoveOverride				: INT := 100;
	fPunchOverride				: INT := 100;

	fThresholdX					: LREAL := -1;
	fThresholdY					: LREAL := -1;
	
	bOutletbelt					: BOOL := TRUE;
	nOutletbeltIntervall		: UINT := 120;
	                    	
	// Toolconfiguration
	stTool						: ST_Tool;	
	stToolHolder				: ST_ToolHolder;
	
	// Holes
	astElements					: ARRAY[0..MATELEMENTS_COUNT] OF ST_Element;
	
END_STRUCT
END_TYPE

// ---- Components/Mat/Structures/ST_Tool.TcDUT
TYPE ST_Tool :
STRUCT
	// Info
	nToolNr						: UINT;
	stToolName					: STRING;
	sNotice						: T_MAXSTRING;
	                        	
	// Geometry             	
	eDieGeometry				: E_Geometry;	
	fLength						: REAL;
	fWidth						: REAL;	
	fRoundCorner				: REAL;
	fRadius						: REAL;
	
END_STRUCT
END_TYPE

// ---- Components/Mat/Structures/ST_ToolHolder.TcDUT
TYPE ST_ToolHolder :
STRUCT
	// Info
	nToolHolderNr				: UINT;
	sToolHolderName				: STRING;
	sToolExtensionNr			: UINT;
	sToolExtensionName			: STRING;
	sNotice						: T_MAXSTRING;
	                        	
	// First Die  	
	bRotateDie					: BOOL;
	fX_Offset					: REAL;
	fY_Offset					: REAL;
	                        	
	// Multi Die            	
	bMultiDie					: BOOL;
	nDieCount					: UINT;
	fDie_Offset					: REAL;
	                        	
END_STRUCT
END_TYPE

// ---- Components/Mat/Structures/ST_Coordinate.TcDUT
TYPE ST_Coordinate :
STRUCT
	fX				: REAL;
	fY				: REAL;
END_STRUCT
END_TYPE

// ---- Components/PunchEngine/Enumerations/E_PunchEngineCmd.TcDUT
{attribute 'qualified_only'}
{attribute 'strict'}
TYPE E_PunchEngineCmd :
(
	cmdNone 	:= 0,
	cmdMove 	:= 1,
	cmdHalt 	:= 2,
	cmdPunch    := 3,
	cmdHome     := 4,
	cmdJog		:= 5
);
END_TYPE

// ---- Machine/Components/E_Axis.TcDUT
/// Enumeration of all axis drives.
TYPE E_Axis :
(
	eAxis_X					:= 0 ,
	eAxis_Y					:= 1 ,
	eAxis_Punch				:= 2 ,

	
	// IMPORTANT: last entry
	eAxis_max
);
END_TYPE

// ---- Machine/Components/E_DigitalOutput.TcDUT
/// Enumeration of all axis drives.
TYPE E_DigitalOutput :
(
	eDigitalOutput_OutletBelt					:= 0 ,

	
	// IMPORTANT: last entry
	eDigitalOutput_max
);
END_TYPE

// ---- Machine/Components/E_Cylinder.TcDUT
/// Enumeration of all Cylinder
TYPE E_Cylinder :
(
	eCylinder_Toolselector					:= 0,

	
	// IMPORTANT: last entry
	eCylinder_max
);
END_TYPE

// ---- Machine/Enumerations/E_JobState.TcDUT
{attribute 'qualified_only'}
{attribute 'strict'}
TYPE E_JobState :
(
	eJobState_none := 0,
	eJobState_ready := 1,
	eJobState_stopped := 2,
	eJobState_running := 3,
	eJobState_error := 4,
	eJobState_finished := 5,
	eJobState_aborted := 6
);
END_TYPE

// ---- Machine/Enumerations/E_MachineArea.TcDUT
/// Enumeration of all possible component types
TYPE E_MachineArea :
(
	/// Common machine part
	eMachineArea_none := 0,
	eMachineArea_common,

	eMachineArea_max
);
END_TYPE

// ---- Machine/Enumerations/E_OperationMode.TcDUT
/// Auflistung aller Betriebsmodi
TYPE E_OperationMode :
(
	eOperationMode_none := 0,
	eOperationMode_Start := 1,
	eOperationMode_Stop  := 2,
	eOperationMode_Halt  := 3,
	eOperationMode_Resume  := 4,
	eOperationMode_Reset  := 5,
	eOperationMode_Maintenance  := 6,
	eOperationMode_Emergency  := 7
);
END_TYPE

// ---- Machine/Enumerations/E_RunTodo.TcDUT
{attribute 'qualified_only'}
{attribute 'strict'}
TYPE E_RunTodo :
(
	Punch_no	 := 0,
	Punch_Tool_1 := 1,
	Punch_Tool_2 := 2
);
END_TYPE

// ---- Machine/Structures/ST_MachineConfig.TcDUT
TYPE ST_MachineConfig :
STRUCT
	fSaftyDistanceToMat					: REAL;	
	
	stMaintPosition						: ST_Coordinate;
	stMaintPositionAlt					: ST_Coordinate;
	stMatOrigin							: ST_Coordinate;
	
	fMoveOutside						: LREAL;
	fPassDistance						: LREAL;
	
	fVelocityX							: LREAL;
	fAccelerationX						: LREAL;
	
	fVelocityY							: LREAL;
	fAccelerationY						: LREAL;
	
	fVelocityPunch						: LREAL;
	fAccelerationPunch					: LREAL;
	
	nPunchTorqueLimit					: INT;
	nPunchTorqueLimitPos				: INT;
	nPunchTorqueLimitNeg				: INT;
	nXTorqueLimit						: INT;
	nYTorqueLimit						: INT;
	
END_STRUCT
END_TYPE

// ---- Machine/Structures/ST_PunchJob.TcDUT
TYPE ST_PunchJob :
STRUCT             	
	Tool_1							: STRING;
	Tool_2							: STRING;
	ToolHolder_1					: STRING;
	ToolHolder_2					: STRING;		
	stMatOffset						: ST_Coordinate;
	
	astRunTodo						: ARRAY[0..MATRUNS_COUNT] OF INT;
	abMultipleMats					: ARRAY[0..MATS_COUNT] OF BOOL;
END_STRUCT
END_TYPE

// ---- Utilities/Component/Enumerations/E_ComponentState.TcDUT
/// Enumeration of all possible (sub) component states
TYPE E_ComponentState :
(
	/// Component state not set
	eComponentState_none := 0,
	/// Component is resetting
	eComponentState_resetting,
	/// Component is ready
	eComponentState_ready,
	/// Component is running
	eComponentState_running,
	/// Component has error
	eComponentState_error
);
END_TYPE

// ---- Utilities/Sequencer/Enumeration/E_SequenceState.TcDUT
/// Auflistung aller Sequence-Stati
TYPE E_SequenceState :
(
	/// Status nicht gesetzt
	eSequenceState_none := 0,
	/// Sequence läuft
	eSequenceState_running,
	/// Sequence wartet im Schritt
	eSequenceState_waiting,
	/// Sequence fertig/ok
	eSequenceState_finished,
	/// Sequence fehlgeschlagen
	eSequenceState_error
);
END_TYPE

// ---- Utilities/TaskAllocation/Enumerations/E_Task.TcDUT
/// Enumeration of all supported PLC Tasks.
TYPE E_Task :
(
	/// Default PLC Task
	eTask_main := 0,
	/// Fast Task
	eTask_fast,
	/// Slow Task
	eTask_slow,
	
	
	eTask_max
);
END_TYPE

// ---- Visualisation/Structures/ST_MaintCmds.TcDUT
TYPE ST_MaintCmds :
STRUCT
	bJogXFw				: BOOL;
	bJogXBw				: BOOL;
                    	
	bJogYFw				: BOOL;
	bJogYBw				: BOOL;
		
	bJogPunchFw			: BOOL;
	bJogPunchBw			: BOOL;
	
	bJogOutletBelt		: BOOL;

	bMovePunchBDC		: BOOL;
	bMovePunchTDC		: BOOL;
	bMoveXYMaint		: BOOL;
	bMoveXYMaintAlt		: BOOL;
	
	bLoadConfig			: BOOL;
	
	bReset				: BOOL;
	bSetZero			: BOOL;
	
	bChangeTool			: BOOL;
END_STRUCT
END_TYPE

// ---- Visualisation/Structures/ST_MaintParam.TcDUT
TYPE ST_MaintParam :
STRUCT
	nChangeTool			: INT;
END_STRUCT
END_TYPE

// ---- Visualisation/Structures/ST_PunchCmds.TcDUT
TYPE ST_PunchCmds :
STRUCT
	bStart					: BOOL;
	bLoad					: BOOL;
	bStop					: BOOL;
	bResume					: BOOL;
	bHalt					: BOOL;
	bOverride				: BOOL;
	
	bLoadLeft				: BOOL;
	bLoadRight				: BOOL;
	bLoadStop				: BOOL;
	bUnlock					: BOOL;
	bMoveTDC				: BOOL;
	bOutletBelt				: BOOL;
END_STRUCT
END_TYPE

// ---- Visualisation/Structures/ST_PunchInfo.TcDUT
TYPE ST_PunchInfo :
STRUCT
	sCleartext				: STRING;
	
	nCurRun					: UINT;
	nCurPunch				: UDINT;
	nCurMat					: UINT;
	
	nMaxPunches				: UDINT;
	
	nCountRemainHolesOfJob	: UDINT;
	nCountAllHolesOfJob		: UDINT;
	nRemainTimeOfJob		: UDINT;
	
	stCoordinate			: ST_Coordinate;	
	bResumeAllowed			: BOOL;
	bPunching				: BOOL;
	eJobState				: E_JobState;
	
	fOverride				: LREAL;
	fPunchspeed				: LREAL;
	
	bLocked					: BOOL;
	
END_STRUCT
END_TYPE

// ---- Visualisation/Structures/ST_MaintInfo.TcDUT
TYPE ST_MaintInfo :
STRUCT	
	// X - Axis
	bXHomed					: BOOL;
	bXError					: BOOL;
	bXMoving				: BOOL;
	fXPosition				: LREAL;
	fXTemp					: LREAL;
	fXMotorTemp				: LREAL;	
	
	// Y - Axis
	bYHomed					: BOOL;
	bYError					: BOOL;
	bYMoving				: BOOL;
	fYPosition				: LREAL;
	fYTemp					: LREAL;
	fYMotorTemp				: LREAL;
	
	// Punch - Axis
	bPunchHomed				: BOOL;
	bPunchError				: BOOL;
	bPunchMoving			: BOOL;
	fPunchPosition			: LREAL;	
	fPunchTemp				: LREAL;
	fPunchMotorTemp			: LREAL;
	nPunchCount				: UDINT;
	
	// ToolChanger
	bToolError				: BOOL;
	bToolChanged			: BOOL;
	nToolSelect				: INT;
	
	// Machine 
	bSequenceError			: BOOL;
	bSafetyOk				: BOOL;	
	bEmergency				: BOOL;
	bSafetyDoor				: BOOL;
	nStep					: INT;
	nSequence				: INT;
	
END_STRUCT
END_TYPE

// ---- Visualisation/Structures/ST_PunchParam.TcDUT
TYPE ST_PunchParam :
STRUCT		
	fOverride				: LREAL;
	bCheckPosBeforeRun		: BOOL;
END_STRUCT
END_TYPE

// ---- BaseComponents/Supervision/GVL_Supervision.TcGVL
{attribute 'qualified_only'}
VAR_GLOBAL
	
	/// GENERAL
	aCodeErr						: ARRAY[0..eCodeError_maxIdx] OF BOOL;
	 
END_VAR

// ---- Machine/Components/COMP_CONST.TcGVL
VAR_GLOBAL CONSTANT
	
	/// Zero based max index for axis
	nMaxIdxAxis						: INT := eAxis_max - 1;
	nMaxIdxCylinder					: INT := eCylinder_max - 1;	
	nMaxIdxDigitalOutput			: INT := eDigitalOutput_max - 1;	
	
END_VAR

// ---- Machine/Components/COMP.TcGVL
VAR_GLOBAL
	
	/// Linked Safety
	{attribute 'TcContextName':='IOTask'}
	stSafetyIO						: ST_SafetyIO;

	/// Linked EtherCAT state
	{attribute 'TcContextName':='IOTask'}
	stEtherCATState					: ST_EtherCatIO;	
	
	/// Linked Component
	{attribute 'TcContextName' := 'IOTask'}
	aStCylinderIO					: ARRAY[0..COMP_CONST.nMaxIdxCylinder] OF ST_CylinderDriverIO;
	{attribute 'TcContextName' := 'IOTask'}
	aStDigitalOutputIO				: ARRAY[0..COMP_CONST.nMaxIdxDigitalOutput] OF ST_DigitalOutputIO;
	{attribute 'TcContextName':='IOTask'}
	stSafetyLockIO					: ST_SafetyLockIO;
		
	
	/// Linked Axis
	{attribute 'TcContextName' := 'NcTask'}
	astAxisRef						: ARRAY[0..COMP_CONST.nMaxIdxAxis] OF AXIS_REF;
	{attribute 'TcContextName' := 'NcTask'}
	astAxisIO						: ARRAY[0..COMP_CONST.nMaxIdxAxis] OF ST_AxisIO;

END_VAR

// ---- Machine/GVL.TcGVL
VAR_GLOBAL
	// Eventlog
	fbEventLog						: FB_Eventlog;	

	// System
	fbSafety						: FB_Safety;
	fbEtherCATBus					: FB_EtherCATBus;
	fbSupervision					: FB_Supervision;	
	
	// Hardware
	fbSafetyLock					: FB_SafetyLock;
	fbMat							: FB_Mat;
	fbPunchEngine					: FB_PunchEngine;
	fbMatAndToolHandling			: FB_MatAndToolHandling;
END_VAR

// ---- Machine/GVL_CONST.TcGVL
VAR_GLOBAL CONSTANT	
	/// GENERAL
	nMaschineID						: INT := 1;
	bActive 						: BOOL := TRUE;
	sName 							: STRING := 'PunchingMachine';
		
	
	/// VALUES, LIMITS          
	MATS_COUNT						: UINT := 3; 			
	MATRUNS_COUNT					: UINT := 7;
	MATELEMENTS_COUNT				: UINT := 32;
	MATHOLES_COUNT					: UINT := 65535;
	
	fEpsilon						: LREAL := 1E-2;	
	tMaxTime						: TIME := T#71582M47S295MS;
	iMaxIdxComponent				: INT := 255;
	iMaxIdxEvents					: INT := eEvent_Max - 1;
	
			
	/// COLORS
	colBlack						: DWORD := 16#FF000000;
	colWhite						: DWORD := 16#FFFFFFFF;
	coldarkGrey						: DWORD := 16#FF505050;
	collmidGrey						: DWORD := 16#FFE6E6E6;
	collightGrey					: DWORD := 16#FFE6E6E6;
	colYellow						: DWORD := 16#FFFFFF00;
	colGreen						: DWORD := 16#FFADE204;
	colOrange						: DWORD := 16#FFFFA500;
	colBlue							: DWORD := 16#FF0000FF;
	colRed							: DWORD := 16#FFFF0000;			
	colSemiBlack					: DWORD := 16#7F000000;
	colSemiWhite					: DWORD := 16#7FFFFFFF;
	colSemidarkGrey					: DWORD := 16#7F505050;
	colSemilmidGrey					: DWORD := 16#7FE6E6E6;
	colSemilightGrey				: DWORD := 16#7FE6E6E6;
	colSemiYellow					: DWORD := 16#7FFFFF00;
	colSemiGreen					: DWORD := 16#7FADE204;
	colSemiOrange					: DWORD := 16#7FFFA500;
	colSemiBlue						: DWORD := 16#7F0000FF;
	colSemiRed						: DWORD := 16#7FFF0000;	 

END_VAR

// ---- Visualisation/GVL_VISU.TcGVL
VAR_GLOBAL
	init_ST_TOOL			: ST_TOOL;
	init_ST_TOOLHOLDER		: ST_TOOLHOLDER;
	init_ST_MAT				: ST_MAT;
	init_ST_MATRUN			: ST_MATRUN;
	init_ST_ELEMENT			: ST_ELEMENT;
	init_ST_PunchJob		: ST_PunchJob;
	init_ST_PunchCmds		: ST_PunchCmds;
	init_ST_PunchInfo		: ST_PunchInfo;
	init_ST_Config			: ST_MachineConfig;
	
	stMaintCmds				: ST_MaintCmds;	
	stMaintParam			: ST_MaintParam;	
	stMaintInfo				: ST_MaintInfo;	
	
	stPunchCmds				: ST_PunchCmds;	
	stPunchParam			: ST_PunchParam;
	stPunchInfo				: ST_PunchInfo;

	stMachineConfig			: ST_MachineConfig;	
	stCurMat				: ST_Mat;
	stPunchJob				: ST_PunchJob;		
END_VAR

// ---- BaseComponents/AxisDriver/Interfaces/ITFMotionComponent.TcIO
INTERFACE ITFMotionComponent EXTENDS ITFComponent

PROPERTY PUBLIC ActPos : LREAL
GET
END_GET
END_PROPERTY

/// Get's the axis reference
PROPERTY Axis : AXIS_REF
GET
END_GET
END_PROPERTY

/// Get`s the MC axis state.
PROPERTY AxisState : ST_AxisStatus
GET
END_GET
END_PROPERTY

PROPERTY Enable : BOOL
GET
END_GET
SET
END_SET
END_PROPERTY

PROPERTY EnableNeg : BOOL
GET
END_GET
SET
END_SET
END_PROPERTY

PROPERTY EnablePos : BOOL
GET
END_GET
SET
END_SET
END_PROPERTY

/// Axis halt using default parameter
{attribute 'object_name' := 'Halt'}
METHOD Halt : E_OperationResult
END_METHOD

PROPERTY Override : LREAL
GET
END_GET
SET
END_SET
END_PROPERTY

PROPERTY Velocity : LREAL
GET
END_GET
END_PROPERTY

END_INTERFACE

// ---- BaseComponents/CylinderDriver/Interfaces/ITF_Cylinder.TcIO
INTERFACE ITF_Cylinder EXTENDS ITFComponent

PROPERTY PUBLIC ActualPosition : E_CylinderPosition
GET
END_GET
END_PROPERTY

PROPERTY PUBLIC EnableHp : BOOL
GET
END_GET
SET
END_SET
END_PROPERTY

PROPERTY PUBLIC EnableWp : BOOL
GET
END_GET
SET
END_SET
END_PROPERTY

// Ansteuerzeit für Impulsventile (0 deaktiviert die Impulssteuerung)
PROPERTY PUBLIC ImpulseTime : TIME
GET
END_GET
SET
END_SET
END_PROPERTY

/// Verweilzeit bis die jeweilige Endlage bestätigt wird.
PROPERTY PUBLIC PositionValidationTime : TIME
GET
END_GET
SET
END_SET
END_PROPERTY

METHOD PUBLIC ResetValves
VAR_INPUT
END_VAR
END_METHOD

PROPERTY PUBLIC SafetyOk : BOOL
GET
END_GET
SET
END_SET
END_PROPERTY

PROPERTY PUBLIC SensorHp : BOOL
GET
END_GET
END_PROPERTY

PROPERTY PUBLIC SensorWp : BOOL
GET
END_GET
END_PROPERTY

/// Verweilzeit nach Ventilansteuerung, bis die Zylinderendlage geprüft wird (0 deaktiviert die Überwachung)
PROPERTY PUBLIC SupervisionTime : TIME
GET
END_GET
SET
END_SET
END_PROPERTY

METHOD PUBLIC ToHP
VAR_INPUT
END_VAR
END_METHOD

METHOD PUBLIC ToWP
VAR_INPUT
END_VAR
END_METHOD

END_INTERFACE

// ---- Utilities/Component/Interfaces/ITFComponent.TcIO
INTERFACE ITFComponent EXTENDS __SYSTEM.IQueryInterface

/// Get's or set's a value indicating whether this component is active or not.
PROPERTY Active : BOOL
GET
END_GET
SET
END_SET
END_PROPERTY

PROPERTY BMK : STRING
GET
END_GET
SET
END_SET
END_PROPERTY

/// Get's value representing the component state.
PROPERTY ClearText : String
GET
END_GET
END_PROPERTY

PROPERTY ID : INT
GET
END_GET
SET
END_SET
END_PROPERTY

/// Get's value representing the component state.
PROPERTY LastError : STRING
GET
END_GET
END_PROPERTY

PROPERTY MachineArea : E_MachineArea
GET
END_GET
SET
END_SET
END_PROPERTY

PROPERTY Name : STRING
GET
END_GET
SET
END_SET
END_PROPERTY

PROPERTY Path : String
GET
END_GET
END_PROPERTY

/// Reset component logic
{attribute 'object_name' := 'Reset'}
METHOD Reset
END_METHOD

/// Run component logic
{attribute 'object_name' := 'Run'}
METHOD Run : E_ComponentState
END_METHOD

/// Set HMI reference
METHOD SetEventLogReference
VAR_IN_OUT
	/// HMI access provider.
	fbEventLogRef	: FB_EventLog;
END_VAR
END_METHOD

/// Get's value representing the component state.
PROPERTY State : E_ComponentState
GET
END_GET
END_PROPERTY

/// Get's value representing the component state.
PROPERTY StateAsString : STRING
GET
END_GET
END_PROPERTY

PROPERTY Typ : E_ComponentType
GET
END_GET
END_PROPERTY

END_INTERFACE

// ---- Utilities/TaskAllocation/Interfaces/ITF_TaskAllocation.TcIO
INTERFACE ITF_TaskAllocation

METHOD Invoke
VAR_INPUT
END_VAR
END_METHOD

PROPERTY Task : E_Task
GET
END_GET
SET
END_SET
END_PROPERTY

PROPERTY TaskId : Int
GET
END_GET
SET
END_SET
END_PROPERTY

END_INTERFACE

// ---- Machine/P_Machine.TcPOU
PROGRAM P_Machine 

VAR	
	// MachineConfig
	stCurMachineConfig				: ST_MachineConfig;
	fOverride						: LREAL;
	bCheckPosBeforeRun				: BOOL;
	
	/// Sequences	
	seqOpMode						: FB_Sequence;
	
	bMaintMat						: BOOL;
	bMaintTool						: BOOL;
	stPunchJob						: ST_PunchJob;
		
	/// Components	
	fbComponents					: FB_CompositionBase;

	// PunchParameters
	bMatLoaded						: BOOL;
	bContinuous						: BOOL;
	nCurRun							: UINT;
	nCurPunch						: UDINT;
	nCurMat							: UINT;	
	nCurMoveOverride				: REAL;
	
	fThresholdX						: LREAL;
	fThresholdY						: LREAL;
	
	stCoordinate					: ST_Coordinate;
	stNextCoordinate				: ST_Coordinate;
	nMaxPunches						: UDINT;
	
	fMaxDisplacementX				: LREAL;
	fMaxDisplacementY				: LREAL;
	
	bInitialized					: BOOL;
	eJobState						: E_JobState;
	
	rtSafety						: R_TRIG;
	
	bSafeDrive						: BOOL;
	
	
END_VAR

// Init
Init();

bSafeDrive := fbSafety.SafetyOk AND fbSafetyLock.SafetyOk;

rtSafety(CLK:= NOT fbSafety.SafetyOk);

// SAFETY
IF rtSafety.Q THEN
	bInitialized := FALSE;
	seqOpMode.Start(E_OperationMode.eOperationMode_Halt);
	fbEventLog.WriteInfo(E_Event.eEvent_none, 'NOT HALT');
	
	IF eJobState = E_JobState.eJobState_running THEN
		eJobState := E_JobState.eJobState_stopped;
	END_IF
	
END_IF

// Run Components
fbEventLog.Run();
fbComponents.Run();

// Run Sequencer
seqOpMode.Enable := TRUE;
seqOpMode.Base(TRUE,FALSE);
CASE seqOpMode.SequenceId OF	
	E_OperationMode.eOperationMode_Maintenance:		_Maintenance();
	E_OperationMode.eOperationMode_Start:			_Start();
	E_OperationMode.eOperationMode_Stop:			_Stop();
	E_OperationMode.eOperationMode_Reset:			_Reset();
	E_OperationMode.eOperationMode_Halt:			_Halt();
END_CASE

METHOD _Halt : BOOL
VAR_INPUT
END_VAR
seqOpMode.Name := 'Halt';

CASE seqOpMode.Step OF
	
0	 :	seqOpMode.StepDefinition('Move to Zero Position', T#0S);
		fbPunchEngine.Halt();
		fbMatAndToolHandling.Halt();
		seqOpMode.NextStepDelay(T#1S, 10);	
		
10	 :	//fbSafetyLock.Unlock();
		seqOpMode.Finish();
		
END_CASE
END_METHOD

METHOD _Maintenance : BOOL
VAR_INPUT
END_VAR
seqOpMode.Name := 'Maintenance';

CASE seqOpMode.Step OF
	

0	 :	seqOpMode.StepDefinition('Move PunchEngine to Maint Position', T#0S);	
		fbPunchEngine.MoveTDC();			
		fbPunchEngine.OutletBeltseq(FALSE, 0);
		seqOpMode.NextStep(10);
	
10	 :	IF fbPunchEngine.TDC THEN
			seqOpMode.NextStep(20);		
		END_IF
		
20	 :	seqOpMode.StepDefinition('Move XY to Maint Position', T#0S);	
		fbMatAndToolHandling.MaintPos(NOT bMaintMat, NOT bMaintTool);	
		seqOpMode.NextStep(30);			
	
30	 :	IF fbMatAndToolHandling.TargetReached THEN 	
			seqOpMode.Finish();		
			//fbSafetyLock.Unlock();
		END_IF

			
END_CASE
END_METHOD

METHOD _Reset : BOOL
VAR_INPUT
END_VAR
CASE seqOpMode.Step OF

	0:	seqOpMode.StepDefinition('reset, init reset WF', T#0S);
		
		fbSafetyLock.Lock();
		bInitialized := FALSE;
		fbComponents.ResetComponents(FALSE, FALSE, 0, 0);
		
		fbEventLog.Mute := TRUE;
		fbEventLog.Reset();	
		
		seqOpMode.NextStepDelay(T#200MS, 10);	// skip safety

	10:	seqOpMode.StepDefinition('Reset: wait for request', T#0S);
		fbSafety.Reset();
		seqOpMode.NextStep(20);
		
	20:	seqOpMode.StepDefinition('Reset safety', T#0S);
		seqOpMode.NextStepTransition(30, fbSafety.State = E_ComponentState.eComponentState_running);
	
	30:	seqOpMode.StepDefinition('Reset all components', T#0S);
		fbComponents.ResetComponents(FALSE, FALSE, eComponentType_none, eComponentType_Safety);
		seqOpMode.NextStep(40);
		
	40:	seqOpMode.StepDefinition('wait for components ready...', T#0S);
		seqOpMode.NextStepTransitionDelay(fbComponents.CompostitionState = E_ComponentState.eComponentState_running, T#5S,  50);
		
	50:	seqOpMode.StepDefinition('Move to Zero Position', T#0S);
		fbPunchEngine.MoveTDC();
		fbPunchEngine.OutletBeltseq(FALSE, 0);
		seqOpMode.NextStep(60);	
		
	60:	IF fbPunchEngine.TDC THEN
			seqOpMode.NextStep(70);	
		END_IF
			
	70:	seqOpMode.StepDefinition('Finish', T#0S);
		fbEventLog.Mute := FALSE;
		fbEventLog.Reset();
		bInitialized := TRUE;
		seqOpMode.Finish();
		
END_CASE
END_METHOD

METHOD _Start : BOOL
VAR
	fTime				: LREAL;
	stTmpPosition		: ST_Coordinate;
END_VAR
seqOpMode.Name := 'Start';

CASE seqOpMode.Step OF
	
/// MAT LOOP

0	 :	seqOpMode.StepDefinition('Check Mat', T#0S);
		
		fbSafetyLock.Lock();
		IF NOT bInitialized THEN			// AUTO INIT
			seqOpMode.NextSequenceId := eOperationMode_Start;
			seqOpMode.Start(E_operationMode.eOperationMode_Reset);
			RETURN;
		END_IF
		
		IF NOT fbMatAndToolHandling.Ready OR NOT fbPunchEngine.Ready THEN
			RETURN;
		END_IF

		IF nCurMat > MATS_COUNT THEN
			fbPunchEngine.MoveTDC();
			fbMatAndToolHandling.MoveRelX(stCurMachineConfig.fMoveOutside ,stCurMachineConfig.fVelocityX, stCurMachineConfig.fAccelerationX);
			fbEventLog.WriteInfo(E_Event.eEvent_none, 'no further Mat Found');
			seqOpMode.NextStep(5);		
			RETURN;
		END_IF		

		IF stPunchJob.abMultipleMats[nCurMat] THEN
			fbMatAndToolHandling.SetupMat(fbMat.Mat.astMatOrigins[nCurMat]);	
			fbPunchEngine.MoveTDC();
			seqOpMode.NextStep(10);
		ELSE	
			nCurMat:= nCurMat + 1;
		END_IF	
		
5	 :	seqOpMode.StepDefinition('Finish Job', T#0S);
		IF fbMatAndToolHandling.TargetReached AND fbPunchEngine.TDC THEN
			fbPunchEngine.OutletBeltOnce();		
			eJobState := E_JobState.eJobState_finished;
			Halt();
		END_IF
		
10	 :	seqOpMode.StepDefinition('Move PunchEngine to Zero Position', T#0S);
		IF fbPunchEngine.TDC THEN
			seqOpMode.NextStep(20);		
		END_IF

/// RUN LOOP		
		
20	 :	seqOpMode.StepDefinition('Check Run if active', T#0S);		
		IF nCurRun > MATRUNS_COUNT THEN
			fbEventLog.WriteInfo(E_Event.eEvent_none, 'no further Run Found');
			nCurMat:= nCurMat + 1;
			nCurRun := 0;		
			seqOpMode.NextStep(0);
			RETURN;
		END_IF

		CASE stPunchJob.astRunTodo[nCurRun] OF			
			E_RunTodo.Punch_Tool_1:	
				fbMatAndToolHandling.SetupToolholder(1,fbMat.Mat.astRuns[nCurRun].stToolHolder.fX_Offset, fbMat.Mat.astRuns[nCurRun].stToolHolder.fY_Offset);
				fbMatAndToolHandling.ChangeTool(1);
				seqOpMode.NextStep(30);	
			
			E_RunTodo.Punch_Tool_2:	
				fbMatAndToolHandling.SetupToolholder(2,fbMat.Mat.astRuns[nCurRun].stToolHolder.fX_Offset, fbMat.Mat.astRuns[nCurRun].stToolHolder.fY_Offset);
				fbMatAndToolHandling.ChangeTool(2);
				seqOpMode.NextStep(30);		
				
			ELSE
				nCurRun := nCurRun + 1;			
		END_CASE

30	 :	seqOpMode.StepDefinition('Changing Tool', T#0S);
		IF fbMatAndToolHandling.ToolChanged THEN
			seqOpMode.NextStep(40);
		END_IF
		
40	 :	seqOpMode.StepDefinition('Prepare Data of current Run', T#0S);
		nMaxPunches := fbMat.Count_HolesOfRun(nCurRun);			
		fMaxDisplacementX	:= 0;
		fMaxDisplacementY	:= 0;
		
		
		// get Coordiantes of MatRun
		IF fbMat.SortRun(nCurRun) <> E_OperationResult.eOperationResult_Ok THEN		
			fbEventLog.WriteWarning(E_Event.eEvent_none, 'Error while sorting Coordinate-Array', FALSE);
			seqOpMode.Finish();
			RETURN;
		END_IF
				
		IF fbMat.ResortCoordinates(E_CoordinatesSortState.eCoordinatesSortState_resorted_v1) <> E_OperationResult.eOperationResult_Ok THEN
			fbEventLog.WriteWarning(E_Event.eEvent_none, 'Error while resorting Coordinate-Array', FALSE);
			seqOpMode.Finish();
			RETURN;
		END_IF
				

		// Set/Calc Override, Velocity, Acceleratopn of Punch	
		nCurMoveOverride := SEL(fbMat.Mat.astRuns[nCurRun].fMoveOverride = 0, INT_TO_REAL(fbMat.Mat.astRuns[nCurRun].fMoveOverride), 100)/100;
		
		fThresholdX:= SEL(fbMat.Mat.astRuns[nCurRun].fThresholdX = -1, fbMat.Mat.astRuns[nCurRun].fThresholdX, fbMat.MaxDistanceX);
		fThresholdY:= SEL(fbMat.Mat.astRuns[nCurRun].fThresholdY = -1, fbMat.Mat.astRuns[nCurRun].fThresholdY, fbMat.MaxDistanceY);
		fTime := fbMatAndToolHandling.GetMovementTime(  fThresholdX, 
													    fThresholdY,
														stCurMachineConfig.fVelocityX,
														stCurMachineConfig.fAccelerationX*nCurMoveOverride, 
														stCurMachineConfig.fVelocityY,
														stCurMachineConfig.fAccelerationY);	
		fbPunchEngine.SetupPunch(fbMat.Mat.fHeight, stCurMachineConfig.fSaftyDistanceToMat, stCurMachineConfig.fVelocityPunch, stCurMachineConfig.fAccelerationPunch, fTime);
		Override := SEL(fbMat.Mat.astRuns[nCurRun].fPunchOverride = 0, fbMat.Mat.astRuns[nCurRun].fPunchOverride, 100);
		
		// Calculate Coordinates		
		IF fbMat.GetCoordinate(nCurRun, nCurPunch, ADR(stCoordinate)) = E_OperationResult.eOperationResult_NOk THEN
			fbEventLog.WriteWarning(E_Event.eEvent_none, 'Error in getting Coordinate', FALSE);
			seqOpMode.Finish();
			RETURN;
		END_IF	
		
		stCoordinate.fX := stCoordinate.fX + stCurMachineConfig.stMatOrigin.fX;	
		stCoordinate.fY := stCoordinate.fY + stCurMachineConfig.stMatOrigin.fY;		
		
		
		// Move to Coordinate
		stTmpPosition := stCoordinate;
		stTmpPosition.fX := stTmpPosition.fX - stCurMachineConfig.fPassDistance;
		fbMatAndToolHandling.MoveAbs(	stTmpPosition, 
										stCurMachineConfig.fVelocityX, 
										stCurMachineConfig.fAccelerationX, 
										stCurMachineConfig.fVelocityY, 
										stCurMachineConfig.fAccelerationY);	

			
		seqOpMode.NextStep(45);		
		
45	 : 	seqOpMode.StepDefinition('Start from the same Direction', T#0S);
		IF fbMatAndToolHandling.TargetReached THEN
			fbMatAndToolHandling.MoveAbs(	stCoordinate, 
											stCurMachineConfig.fVelocityX, 
											stCurMachineConfig.fAccelerationX*nCurMoveOverride, 
											stCurMachineConfig.fVelocityY, 
											stCurMachineConfig.fAccelerationY);			
			seqOpMode.NextStep(50);		
		END_IF	
			
50	 : 	seqOpMode.StepDefinition('Move to First Position Before Loop', T#0S);
		IF fbMatAndToolHandling.TargetReached AND NOT bCheckPosBeforeRun THEN	
			seqOpMode.NextStep(60);		
		END_IF		
		
		IF seqOpMode.NextSequence THEN
			seqOpMode.Finish();
			RETURN;
		END_IF		
		
// PUNCHING LOOP
	
60	 :	seqOpMode.StepDefinition('Preparing', T#0S);
		IF fbMat.GetCoordinate(nCurRun, nCurPunch, ADR(stCoordinate)) = E_OperationResult.eOperationResult_NOk THEN
			fbEventLog.WriteWarning(E_Event.eEvent_none, 'Error in getting Coordinate', FALSE);
			seqOpMode.Finish();
			RETURN;
		END_IF	
		
		// outletbelt	
		IF fbMat.Mat.astRuns[nCurRun].bOutletbelt THEN
			fbPunchEngine.OutletBeltSeq(TRUE, fbMat.Mat.astRuns[nCurRun].nOutletbeltIntervall);
		END_IF
		
		// get next Coordinate	
		fbMat.GetCoordinate(nCurRun, nCurPunch+1, ADR(stNextCoordinate));
			
		IF seqOpMode.NextSequence THEN
			bContinuous := FALSE;
		ELSIF nCurPunch + 1 >= nMaxPunches THEN
			bContinuous := FALSE;
		ELSIF ABS(stNextCoordinate.fX - stCoordinate.fX) <= (fThresholdX + 0.1)				/// Nummerischer Fehler beim Berechnen des Treshholds wird mit 0.1 ausgeglichen 
		  AND ABS(stNextCoordinate.fY - stCoordinate.fY) <= (fThresholdY + 0.1) THEN
			bContinuous := TRUE;
		ELSE
			bContinuous := FALSE;
		END_IF
		
		// Calculate Asolute Coordinates
		stCoordinate.fX := stCoordinate.fX + stCurMachineConfig.stMatOrigin.fX;
		stCoordinate.fY := stCoordinate.fY + stCurMachineConfig.stMatOrigin.fY;		
		
		// Move to Coordinate
		fbMatAndToolHandling.MoveAbs(	stCoordinate, 
										stCurMachineConfig.fVelocityX, 
										stCurMachineConfig.fAccelerationX*nCurMoveOverride, 
										stCurMachineConfig.fVelocityY, 
										stCurMachineConfig.fAccelerationY);		
										
		IF fbPunchEngine.Punching THEN
			fbPunchEngine.Punch(bContinuous);
			seqOpMode.NextStep(80);	
		ELSE
			seqOpMode.NextStep(70);			
		END_IF	
		
70	 :	seqOpMode.StepDefinition('Moving', T#0S);
		// Anforderung auf Operationsmoduswechsel
		IF seqOpMode.NextSequence THEN
			seqOpMode.Finish();
			RETURN;
		END_IF		


		IF fbMatAndToolHandling.TargetReached THEN	
			fbPunchEngine.Punch(bContinuous);
			seqOpMode.NextStep(80);		
		END_IF		
		
80	 :	seqOpMode.StepDefinition('Punching', T#0S);

		// Wenn nicht durchgehend gestanzt wird warten bis der Stanzprozess abgeschlossen ist
		IF NOT bContinuous AND fbPunchEngine.Punching THEN
			RETURN;
		END_IF
	
		// Überprüfe den Unterschied zwischen IST/SOLL Position -> FEHLER bei zu hohem Unterschied
		IF fbPunchEngine.PunchDone THEN		
			stTmpPosition := fbMatAndToolHandling.Position;
			fMaxDisplacementX := MAX(fMaxDisplacementX, ABS(stCoordinate.fX - stTmpPosition.fX));
			fMaxDisplacementY := MAX(fMaxDisplacementY, ABS(stCoordinate.fY - stTmpPosition.fY));	
			nCurPunch := nCurPunch + 1;
			seqOpMode.NextStep(60);	
		END_IF
		
		// Keine weitere Stanzung in diesem Durchgang 
		IF nCurPunch >= nMaxPunches THEN
			fbEventLog.WriteInfo(E_Event.eEvent_none, 'Run Finished');
			fbPunchEngine.OutletBeltSeq(FALSE, 0);
			nCurPunch := 0;
			nCurRun := nCurRun + 1;
			seqOpMode.NextStep(20);	
			RETURN;
		END_IF	
		

END_CASE
END_METHOD

METHOD _Stop : BOOL
VAR_INPUT
END_VAR
seqOpMode.Name := 'Stop';

CASE seqOpMode.Step OF
	
0	 :	seqOpMode.StepDefinition('Move Punch to Zero Position', T#0S);
		fbPunchEngine.MoveTDC();
		fbPunchEngine.OutletBeltOnce();
		seqOpMode.NextStep(10);	
		
10	 :	seqOpMode.StepDefinition('Move Punch to Zero Position', T#0S);	
		IF fbPunchEngine.TDC THEN
			seqOpMode.NextStep(20);	
		END_IF
	
20	 :	seqOpMode.StepDefinition('Move Y-Axis to Zero Position', T#0S);		
		fbMatAndToolHandling.MoveAbsY(10, stCurMachineConfig.fVelocityX, stCurMachineConfig.fAccelerationX); //TODO: not hardcoded Position
		seqOpMode.NextStep(30);	

30	 :  IF fbMatAndToolHandling.TargetReached THEN
			fbPunchEngine.OutletBeltOnce();	
			seqOpMode.NextStepDelay(T#1S, 40);	
		END_IF	
		
40	 :	seqOpMode.StepDefinition('Stop finished', T#0S);	
		//fbSafetyLock.Unlock();
		seqOpMode.Finish();
		
	
END_CASE
END_METHOD

PROPERTY CheckPosBeforeRun : BOOL
GET
CheckPosBeforeRun := bCheckPosBeforeRun;
END_GET
SET
bCheckPosBeforeRun := CheckPosBeforeRun;
END_SET
END_PROPERTY

METHOD ClearJob : BOOL
VAR_INPUT
END_VAR
nCurRun := 0;
nCurPunch := 0;
nCurMat := 0;
MEMSET(ADR(stPunchJob), 0, SIZEOF(stPunchJob));

eJobState := E_JobState.eJobState_none;
END_METHOD

PROPERTY CountAllHolesOfJob : UDINT
GET
VAR
	ni						: UINT;
	nMats					: UINT;
	nPunchCount				: UDINT;
END_VAR
IF NOT bMatLoaded THEN
	RETURN;
END_IF

nMats := 0;
FOR ni := 0 TO MATS_COUNT DO
	IF 	stPunchJob.abMultipleMats[ni] THEN
		nMats := nMats + 1;
	END_IF
END_FOR

IF nMats = 0 THEN
	RETURN;
END_IF

nPunchCount := 0;
FOR ni := 0 TO MATRUNS_COUNT DO
	IF stPunchJob.astRunTodo[ni] = 0 THEN
		CONTINUE;
	END_IF
	nPunchCount := nPunchCount + fbMat.Count_HolesOfRun(ni);
END_FOR

CountAllHolesOfJob := nPunchCount * nMats;
END_GET
END_PROPERTY

PROPERTY CountRemainHolesOfJob : UDINT
GET
VAR
	ni						: UINT;
	nMats					: UINT;
	nPunchCount				: UDINT;
END_VAR
IF NOT bMatLoaded THEN
	RETURN;
END_IF

nMats := 0;
FOR ni := nCurMat TO MATS_COUNT DO
	IF 	stPunchJob.abMultipleMats[ni] THEN
		nMats := nMats + 1;
	END_IF
END_FOR

IF nMats = 0 THEN
	RETURN;
END_IF

nPunchCount := 0;
FOR ni := nCurRun TO MATRUNS_COUNT DO
	IF stPunchJob.astRunTodo[ni] = 0 THEN
		CONTINUE;
	END_IF
	nPunchCount := nPunchCount + fbMat.Count_HolesOfRun(ni);
END_FOR

CountRemainHolesOfJob := nPunchCount * nMats - nCurPunch;
END_GET
END_PROPERTY

PROPERTY CurMat : UINT
GET
CurMat := nCurMat;
END_GET
END_PROPERTY

PROPERTY CurPunch : UDINT
GET
CurPunch := nCurPunch;
END_GET
END_PROPERTY

PROPERTY CurRun : UINT
GET
CurRun := nCurRun;
END_GET
END_PROPERTY

METHOD Halt : E_OperationResult
VAR_INPUT
END_VAR
Halt := E_OperationResult.eOperationResult_NOk;

//ClearJob();
seqOpMode.Start(E_OperationMode.eOperationMode_Halt);

Halt := E_OperationResult.eOperationResult_Ok;
END_METHOD

METHOD Init : BOOL
VAR
	stLogConfig						: ST_LoggingConfig;
	stPlcAppSystemInfo				: PlcAppSystemInfo;
END_VAR

VAR_STAT
	OnlineChangesMirror				: UDINT;		
	FirstRun						: BOOL := TRUE;
END_VAR
//Init on OnlineChange
stPlcAppSystemInfo := Statics.stPlcSystemInfo.stPlcAppSystemInfo;
IF OnlineChangesMirror <> stPlcAppSystemInfo.OnlineChangeCnt OR FirstRun THEN
	OnlineChangesMirror := stPlcAppSystemInfo.OnlineChangeCnt;
	FirstRun := FALSE;
	
	InitComponents();
	InitConfig();

END_IF
END_METHOD

METHOD InitComponents : BOOL
VAR
	stLogConfig						: ST_LoggingConfig;
END_VAR
// Eventlog
stLogConfig.eLoggingProvider := E_LoggingProvider.eLoggingProviderEventLog;	
stLogConfig.sLogName := 'Punch.log';	
stLogConfig.sLogPath := 'C:\Log\Punch';									
stLogConfig.eLogLevel := E_LogLevel.eLogLevelInformation; 				
fbEventLog.Config := stLogConfig;
fbEventLog.Reset();

fbComponents.LoadComponents();	
fbComponents.Active := TRUE;
fbComponents.Name := 'Collection of all Components';
fbComponents.SetEventLogReference(fbEventLog);	

/// Supervison
fbComponents.RegisterComponent(1, fbSupervision);
fbSupervision.Active := TRUE;
fbSupervision.Name := 'Supervision';
fbSupervision.MachineArea := .eMachineArea_common;

/// Ethercat-Bus
fbComponents.RegisterComponent(2, fbEtherCATBus);
fbEtherCATBus.Active := TRUE;
fbEtherCATBus.Name := 'EtherCAT Bus';
fbEtherCATBus.MachineArea := E_MachineArea.eMachineArea_common;
fbEtherCATBus.SetReferences(COMP.stEtherCATState);

/// Safety
fbComponents.RegisterComponent(3, fbSafety);
fbSafety.Active := TRUE;
fbSafety.Name := 'Safety';
fbSafety.MachineArea := E_MachineArea.eMachineArea_common;
fbSafety.SetReferences(COMP.stSafetyIO);

/// Mat
fbComponents.RegisterComponent(5, fbMat);
fbMat.Active := TRUE;
fbMat.Name := 'Mat Definition';
fbMat.MachineArea := E_MachineArea.eMachineArea_common;

/// Mat and Tool Handling
fbComponents.RegisterComponent(6, fbMatAndToolHandling);
fbMatAndToolHandling.Active := TRUE;
fbMatAndToolHandling.Name := 'Mat and Tool Handling';
fbMatAndToolHandling.MachineArea := E_MachineArea.eMachineArea_common;
fbMatAndToolHandling.Setup(E_Axis.eAxis_X, E_Axis.eAxis_Y, E_Cylinder.eCylinder_Toolselector);
//fbMatAndToolHandling.Override := 100;
fbMatAndToolHandling.SetupToolDistance(0, 278.7);
fbMatAndToolHandling.SetupEnable(bSafeDrive);

/// Punch Engine
fbComponents.RegisterComponent(4, fbPunchEngine);
fbPunchEngine.Active := TRUE;
fbPunchEngine.Name := 'Punch Engine';
fbPunchEngine.MachineArea := E_MachineArea.eMachineArea_common;
fbPunchEngine.Setup(E_Axis.eAxis_Punch, E_DigitalOutput.eDigitalOutput_OutletBelt);
//fbPunchEngine.Override := 100;
fbPunchEngine.SetupCrank(420, 20);
fbPunchEngine.SetupEnable(bSafeDrive);


/// Safety Lock
fbComponents.RegisterComponent(4, fbSafetyLock);
fbSafetyLock.Active := TRUE;
fbSafetyLock.Name := 'Punch Engine';
fbSafetyLock.MachineArea := E_MachineArea.eMachineArea_common;
fbSafetyLock.SetReferences(COMP.stSafetyLockIO);

Override := 10;

/// Add Log
fbEventLog.Logger.AddLog('System startup, configuration loaded.', sName, E_LogLevel.eLogLevelInformation);
END_METHOD

METHOD InitConfig : BOOL
VAR
	stConfig				: ST_MachineConfig;
END_VAR
stConfig.stMatOrigin.fX := -20.5;
stConfig.stMatOrigin.fY := 343.5;

stConfig.fAccelerationX := 11000;//5500/2;
stConfig.fAccelerationY := 11000;//11000/2;
stConfig.fAccelerationPunch := 11000;

stConfig.fVelocityX := 660;
stConfig.fVelocityY := 660;
stConfig.fVelocityPunch := 900;

stConfig.fSaftyDistanceToMat := 0;

stConfig.stMaintPosition.fX := 10;
stConfig.stMaintPosition.fY := 10;
stConfig.stMaintPositionAlt.fX := 4050;
stConfig.stMaintPositionAlt.fY := 10;

stConfig.fMoveOutside := 440;
stConfig.fPassDistance := 2;

stConfig.nPunchTorqueLimit := 100;
stConfig.nPunchTorqueLimitNeg := 20;
stConfig.nPunchTorqueLimitPos := 100;

stConfig.nXTorqueLimit := 50;
stConfig.nYTorqueLimit := 100;

LoadConfig(stConfig);
END_METHOD

PROPERTY JobState : E_Jobstate
GET
VAR
	ni						: UINT;	
	bCheck					: BOOL;
END_VAR
JobState := eJobState;

//JobState := E_JobState.eJobState_error;
//
//// check if there ist at least one Mat enabled
//bCheck := FALSE;
//FOR ni := 0 TO MATS_COUNT DO
//	IF 	stPunchJob.abMultipleMats[ni] THEN
//		bCheck := TRUE;
//		EXIT;
//	END_IF
//	CONTINUE;
//END_FOR
//IF NOT bCheck THEN
//	RETURN;
//END_IF
//
//// check if there ist at least one Run enabled
//bCheck := FALSE;
//FOR ni := 0 TO MATRUNS_COUNT DO	
//	IF stPunchJob.astRunTodo[ni] <> 0 THEN
//		bCheck := TRUE;
//		EXIT;
//	END_IF
//	CONTINUE;
//END_FOR
//IF NOT bCheck THEN
//	RETURN;
//END_IF
//
//// check differences between Todolist and mat
//FOR ni := 0 TO MATRUNS_COUNT DO
//	IF stPunchJob.astRunTodo[ni] <> 0 AND NOT fbMat.Mat.astRuns[ni].bActive THEN
//		RETURN;
//	END_IF
//END_FOR
//
//
//JobState := E_JobState.eJobState_ready;
//
//IF seqOpMode.SequenceId = eOperationMode_Start AND seqOpMode.State = eSequenceState_running THEN
//	JobState := E_JobState.eJobState_running;
//END_IF
//
//IF nCurRun + nCurPunch + nCurMat = 0 THEN
//	JobState := E_JobState.eJobState_stopped;
//END_IF
END_GET
END_PROPERTY

METHOD LoadConfig : E_OperationResult
VAR_INPUT
	stConfig				: ST_MachineConfig;
END_VAR
LoadConfig := E_OperationResult.eOperationResult_NOk;

stCurMachineConfig := stConfig;

fbPunchEngine.TorqueLimit := stCurMachineConfig.nPunchTorqueLimit;
fbPunchEngine.TorqueLimitNeg := stCurMachineConfig.nPunchTorqueLimitNeg;
fbPunchEngine.TorqueLimitPos := stCurMachineConfig.nPunchTorqueLimitPos;

fbMatAndToolHandling.TorqueLimitX := stCurMachineConfig.nXTorqueLimit;
fbMatAndToolHandling.TorqueLimitY := stCurMachineConfig.nYTorqueLimit;

LoadConfig := E_OperationResult.eOperationResult_Ok;
END_METHOD

METHOD LoadJob : E_OperationResult
VAR_INPUT
	PunchJob				: ST_PunchJob;
END_VAR

VAR
	ni						: UINT;	
	bCheck					: BOOL;
END_VAR
LoadJob := E_OperationResult .eOperationResult_NOk;

// CHECK IF SAME
//IF MEMCMP(ADR(PunchJob), ADR(stPunchJob), SIZEOF(ST_PunchJob)) = 0 THEN
//	LoadJob := E_OperationResult .eOperationResult_Ok;
//	RETURN;
//END_IF

IF eJobState = E_JobState.eJobState_running OR eJobState = E_JobState.eJobState_stopped THEN
	RETURN;
END_IF

// check if Mat is loaded
IF NOT bMatLoaded THEN
	RETURN;
END_IF



// check if there ist at least one Mat enabled
bCheck := FALSE;
FOR ni := 0 TO MATS_COUNT DO
	IF 	PunchJob.abMultipleMats[ni] THEN
		bCheck := TRUE;
		EXIT;
	END_IF
	CONTINUE;
END_FOR
IF NOT bCheck THEN
	RETURN;
END_IF

// check if there ist at least one Run enabled
bCheck := FALSE;
FOR ni := 0 TO MATRUNS_COUNT DO	
	IF PunchJob.astRunTodo[ni] <> 0 THEN
		bCheck := TRUE;
		EXIT;
	END_IF
	CONTINUE;
END_FOR
IF NOT bCheck THEN
	RETURN;
END_IF

// check differences between Todolist and mat
FOR ni := 0 TO MATRUNS_COUNT DO
	IF PunchJob.astRunTodo[ni] <> 0 AND NOT fbMat.Mat.astRuns[ni].bActive THEN
		RETURN;
	END_IF
END_FOR

stPunchJob := PunchJob;	
eJobState := E_JobState.eJobState_ready;

LoadJob := E_OperationResult .eOperationResult_Ok;
END_METHOD

METHOD LoadMat : E_OperationResult
VAR_IN_OUT
	Mat						: ST_Mat;
END_VAR
VAR
	bMatOkay				: BOOL;
	ni						: UINT;
END_VAR
LoadMat := E_OperationResult.eOperationResult_NOk;

bMatLoaded := FALSE;
bMatOkay := FALSE;

IF Mat.fLenght = 0 OR Mat.fWidth = 0 THEN
	RETURN;
END_IF

FOR ni := 0 TO MATRUNS_COUNT DO
	
	// check if there is at lest one active Run
	IF  Mat.astRuns[ni].bActive THEN
		bMatOkay := TRUE;
		EXIT;
	END_IF
	
END_FOR

IF NOT bMatOkay THEN
	RETURN;
END_IF

fbMat.LoadMat(Mat);

bMatLoaded := TRUE;
LoadMat := E_OperationResult.eOperationResult_Ok;
END_METHOD

PROPERTY MachineConfig : ST_MachineConfig
GET
MachineConfig := stCurMachineConfig;
END_GET
SET
stCurMachineConfig := MachineConfig;
END_SET
END_PROPERTY

METHOD Maint : E_OperationResult
VAR_INPUT
	Mat				: BOOL;
	Tool			: BOOL;
	Alt				: BOOL;
END_VAR
Maint := E_OperationResult.eOperationResult_NOk;

IF eJobState = E_JobState.eJobState_running THEN
	eJobState := E_JobState.eJobState_stopped;
END_IF
seqOpMode.NextSequenceId := E_OperationMode.eOperationMode_Maintenance;

// load actual Maintposition
IF Alt THEN
	fbMatAndToolHandling.SetupMaintPos(stCurMachineConfig.stMaintPositionAlt);
ELSE
	fbMatAndToolHandling.SetupMaintPos(stCurMachineConfig.stMaintPosition);
END_IF
bMaintMat := Mat;
bMaintTool := Tool;

Maint := E_OperationResult.eOperationResult_Ok;
END_METHOD

PROPERTY MatLoaded : BOOL
GET
MatLoaded := bMatLoaded;
END_GET
END_PROPERTY

PROPERTY MatOriginX : REAL
GET
MatOriginX := stCurMachineConfig.stMatOrigin.fX;
END_GET
SET
stCurMachineConfig.stMatOrigin.fX := MatOriginX;
END_SET
END_PROPERTY

PROPERTY MatOriginY : REAL
GET
MatOriginY := stCurMachineConfig.stMatOrigin.fY;
END_GET
SET
stCurMachineConfig.stMatOrigin.fY := MatOriginY;
END_SET
END_PROPERTY

PROPERTY MaxPunch : UDINT
GET
MaxPunch := nMaxPunches;
END_GET
END_PROPERTY

PROPERTY Override : Lreal
GET
Override := fOverride;
END_GET
SET
fOverride := Override;
fbPunchEngine.Override := Override;
END_SET
END_PROPERTY

PROPERTY Punching : BOOL
GET
Punching := seqOpMode.SequenceId = eOperationMode_Start AND seqOpMode.State = eSequenceState_running ;
END_GET
END_PROPERTY

PROPERTY RemainTimeOfJob : UDINT
GET
IF fbPunchEngine.Velocity = 0 OR fOverride = 0 THEN
	RETURN;
END_IF

IF NOT Punching THEN
	RETURN;
END_IF

RemainTimeOfJob := LREAL_TO_UDINT(CountRemainHolesOfJob/(fbPunchEngine.Velocity/360)/fOverride*100/60);
END_GET
END_PROPERTY

METHOD Reset : E_OperationResult
VAR_INPUT
END_VAR
Reset := E_OperationResult.eOperationResult_NOk;

IF eJobState = E_JobState.eJobState_running THEN
	eJobState := E_JobState.eJobState_stopped;
END_IF
seqOpMode.Start(e_Operationmode.eOperationMode_Reset);

Reset := E_OperationResult.eOperationResult_Ok;
END_METHOD

METHOD Resume : E_OperationResult
VAR_INPUT
END_VAR

VAR
	ni						: UINT;	
	bCheck					: BOOL;
END_VAR
Resume := E_OperationResult.eOperationResult_NOk;

IF eJobState <> E_JobState.eJobState_ready AND eJobState <> E_JobState.eJobState_stopped THEN
	RETURN;
END_IF;;

IF Override = 0 THEN
	RETURN;
END_IF

eJobState := E_JobState.eJobState_running;
seqOpMode.Start(e_Operationmode.eOperationMode_Start);
Resume := E_OperationResult.eOperationResult_Ok;
END_METHOD

PROPERTY ResumeAllowed : BOOL
GET
VAR
	ni						: UINT;	
	bCheck					: BOOL;
END_VAR
ResumeAllowed := TRUE;

IF Punching THEN
	ResumeAllowed := FALSE;
	RETURN;	
END_IF

IF nCurRun + nCurPunch + nCurMat = 0 THEN
	ResumeAllowed := FALSE;
	RETURN;	
END_IF

// check if Mat is loaded
IF NOT bMatLoaded THEN
	ResumeAllowed := FALSE;
	RETURN;
END_IF

// check if there ist at least one Mat enabled
bCheck := FALSE;
FOR ni := 0 TO MATS_COUNT DO
	IF 	stPunchJob.abMultipleMats[ni] THEN
		bCheck := TRUE;
		EXIT;
	END_IF
	CONTINUE;
END_FOR
IF NOT bCheck THEN
	ResumeAllowed := FALSE;
	RETURN;
END_IF

// check if there ist at least one Run enabled
bCheck := FALSE;
FOR ni := 0 TO MATRUNS_COUNT DO	
	IF stPunchJob.astRunTodo[ni] <> 0 THEN
		bCheck := TRUE;
		EXIT;
	END_IF
	CONTINUE;
END_FOR
IF NOT bCheck THEN
	ResumeAllowed := FALSE;
	RETURN;
END_IF

// check differences between Todolist and mat
FOR ni := 0 TO MATRUNS_COUNT DO
	IF stPunchJob.astRunTodo[ni] <> 0 AND NOT fbMat.Mat.astRuns[ni].bActive THEN
		ResumeAllowed := FALSE;
		RETURN;
	END_IF
END_FOR
END_GET
END_PROPERTY

METHOD Start : E_OperationResult
VAR_INPUT
	PunchJob				: ST_PunchJob;
END_VAR

VAR
	ni						: UINT;	
	bCheck					: BOOL;
END_VAR
Start := E_OperationResult.eOperationResult_NOk;

//IF fbSafetyLock.Opened THEN
//	RETURN;
//END_IF

ClearJob();
LoadJob(PunchJob);

IF Override = 0 THEN
	RETURN;
END_IF

eJobState := E_JobState.eJobState_running;
seqOpMode.Start(e_Operationmode.eOperationMode_Start);
Start := E_OperationResult.eOperationResult_Ok;
END_METHOD

METHOD Stop : E_OperationResult
VAR_INPUT
END_VAR
Stop := E_OperationResult.eOperationResult_NOk;

seqOpMode.NextSequenceId := E_OperationMode.eOperationMode_Stop;

IF eJobState = E_JobState.eJobState_running THEN
	eJobState := E_JobState.eJobState_stopped;
END_IF

Stop := E_OperationResult.eOperationResult_Ok;
END_METHOD

END_PROGRAM

// ---- Utilities/Sequencer/FB_Sequence.TcPOU
/// Sequence
FUNCTION_BLOCK FB_Sequence

VAR		
	/// Name of Sequence
	sName				: STRING := 'Aktion';
	/// Actual Sequence-State
	eState				: E_SequenceState;
	
	/// Step Description
	sClearText			: STRING;
	/// Error Description
	sLastError			: STRING;
	
	/// Enable Sequencer
	bEnable				: BOOL;
	
	/// ID of running Sequence
	nSequenceId			: INT;
	/// ID of next Sequence
	nNextSequenceId		: INT;
	/// ID of last Sequence
	nLastSequenceId		: INT;
	
	/// Pause Sequence only stepping is possible
	bPause				: BOOL;	
	/// Single step option
	bStepping			: BOOL;	
	
	/// actual Sequence first call
	bFirstShotSequence	: BOOL;
	/// actual Step first call
	bFirstShotStep		: BOOL;
	/// Step Timeout - flag 
	bTimeoutStep		: BOOL;

	
	/// Actual Stepnumber
	nStep				: INT;	
	
	/// Copy of Step for first shot trigger
	nStepMirror			: INT := -1;
	/// maximum Steptime (0 -> infinity)
	tMaxStepTime		: TIME := T#0S;
	/// Step Timer
	tonStep				: TON;
	/// StepDelay Timer
	tonStepDelay		: TON;
END_VAR

///
/// Sequence - FB Utility.
/// HF/www.asma.at/02.2018
///

METHOD Base
VAR_INPUT
	AutoNextSequence			: BOOL;
	EnableErrorHandling			: BOOL;
END_VAR
// Enabled
IF NOT bEnable THEN
	init();
	RETURN;
END_IF

// Finished
IF eState = eSequenceState_finished THEN
	sClearText := Concat3('Sequence: ', Name, ' finished');
	eState := eSequenceState_none;
END_IF
	
// Ready for New - start automatically
IF eState = eSequenceState_none AND AutoNextSequence THEN
	IF nNextSequenceId <> 0 THEN
		StartNext();	
	END_IF
END_IF

// 1st shot trigger
bFirstShotStep := nStep <> nStepMirror;
bFirstShotSequence := bFirstShotStep AND nStep = 0;
nStepMirror := nStep;

// run timer
tonStep(IN := NOT bFirstShotStep, PT := GVL_CONst.tMaxTime);
tonStepDelay();

IF bFirstShotStep THEN
	tonStepDelay.IN := FALSE;
END_IF

// step timeout
bTimeoutStep := tMaxStepTime > T#1MS AND tonStep.ET > tMaxStepTime;

// error handling
IF NOT EnableErrorHandling THEN
	RETURN;
END_IF

// State Error
IF eState = eSequenceState_error THEN
	IF LastError = sEmpty THEN
	sLastError := Concat8('ERROR ', sName, ' - Seq: ', INT_TO_STRING(nSequenceId), ', Step: ', INT_TO_STRING(nStep), ', StepTime: ', TIME_TO_STRING(tonStep.ET));
	END_IF	
END_IF

// Timeout
IF bTimeoutStep THEN
	eState := eSequenceState_error;
	sLastError := Concat8('TIMEOUT ', sName, ' - Seq: ', INT_TO_STRING(nSequenceId), ', Step: ', INT_TO_STRING(nStep), ', StepTime: ', TIME_TO_STRING(tonStep.ET));
END_IF
END_METHOD

PROPERTY ClearText : STRING
GET
ClearText := sClearText;
END_GET
SET
sClearText := ClearText;
END_SET
END_PROPERTY

PROPERTY Enable : BOOL
GET
Enable := bEnable;
END_GET
SET
bEnable := Enable;
END_SET
END_PROPERTY

METHOD Finish
VAR_INPUT
END_VAR
nStep := 0;
nStepMirror := -1;

nLastSequenceId := nSequenceId;
nSequenceId := 0;
eState := eSequenceState_finished;
END_METHOD

/// aktuelle Sequence wird zum 1. Mal aufgerufen
{attribute 'monitoring':='variable'}
PROPERTY FirstShotSequence : BOOL
GET
FirstShotSequence := bFirstShotSequence;
END_GET
END_PROPERTY

/// aktueller Schritt wird zum 1. Mal aufgerufen
{attribute 'monitoring':='variable'}
PROPERTY FirstShotStep : BOOL
GET
FirstShotStep := bFirstShotStep;
END_GET
END_PROPERTY

/// Schrittschaltwerk - Initialisierung
METHOD Init
VAR_INPUT
END_VAR
nStep := 0;
nStepMirror := -1;

nLastSequenceId := nSequenceId;
nNextSequenceId := 0;
nSequenceId := 0;
eState := eSequenceState_none;
tonStepDelay.IN := FALSE;
END_METHOD

PROPERTY LastError : STRING
GET
LastError := sLastError;
END_GET
END_PROPERTY

PROPERTY LastSequenceId : INT
GET
LastSequenceId := nLastSequenceId;
END_GET
END_PROPERTY

/// Maximale Schirttdauer (0 -> unbegrenzt)
{attribute 'monitoring':='variable'}
PROPERTY MaxStepTime : TIME
GET
MaxStepTime := tMaxStepTime;
END_GET
SET
tMaxStepTime := MaxStepTime;
END_SET
END_PROPERTY

/// Name der Aktion
{attribute 'monitoring':='variable'}
PROPERTY Name : STRING
GET
Name := sName;
END_GET
SET
sName := Name;
END_SET
END_PROPERTY

PROPERTY NextSequence : BOOL
GET
NextSequence := nNextSequenceId <> 0;
END_GET
END_PROPERTY

PROPERTY NextSequenceId : INT
GET
NextSequenceId := nNextSequenceId;
END_GET
SET
nNextSequenceId := NextSequenceId;
END_SET
END_PROPERTY

METHOD NextStep : BOOL
VAR_INPUT
	Step			: INT;
END_VAR
nStep := Step;
END_METHOD

METHOD NextStepDelay : BOOL
VAR_INPUT
	Delay				: TIME;
	NextStep			: INT;
END_VAR
NextStepTransitionDelay(TRUE, Delay, NextStep);
END_METHOD

METHOD NextStepTransition : BOOL
VAR_INPUT
	NextStep			: INT;
	Condition			: BOOL;
END_VAR
NextStepTransitionDelay(Condition, t#0s, NextStep);
END_METHOD

METHOD NextStepTransitionDelay : BOOL
VAR_INPUT
	Condition			: BOOL;
	Delay				: TIME;
	NextStep			: INT;
END_VAR
IF bPause THEN
	sClearText := CONCAT('Paused - ', sClearText);
ELSIF NOT Condition THEN
	sClearText := CONCAT('Waiting - ', sClearText);
END_IF

tonStepDelay.IN := TRUE;
tonStepDelay.PT:= Delay;

IF Condition AND (Delay = T#0S OR tonStepDelay.Q OR bPause) AND (NOT bPause OR bStepping) THEN
	tonStepDelay.IN := FALSE;
	bStepping := FALSE;
	nStep:= NextStep;
END_IF
END_METHOD

METHOD Pause 
VAR_INPUT
	Enable			:bool;
END_VAR
bPause := Enable;
END_METHOD

PROPERTY SequenceId : INT
GET
SequenceId := nSequenceId;
END_GET
END_PROPERTY

METHOD Start
VAR_INPUT
	nId 	: INT;
END_VAR
nStep := 0;
nStepMirror := -1;

nSequenceId := nId;
eState := eSequenceState_running;
END_METHOD

METHOD StartLast
VAR_INPUT
END_VAR
Init();

IF nLastSequenceId <> 0 THEN
	nStep := 0;
	nStepMirror := -1;
	
	nSequenceId := nLastSequenceId;
	eState := eSequenceState_running;
END_IF
END_METHOD

METHOD StartNext
VAR_INPUT
END_VAR
IF nNextSequenceId <> 0 THEN
	nStep := 0;
	nStepMirror := -1;
	
	nSequenceId := nNextSequenceId;
	nNextSequenceId := 0;
	eState := eSequenceState_running;
END_IF
END_METHOD

/// aktueller Sequence-Status
{attribute 'monitoring':='variable'}
PROPERTY State : E_SequenceState
GET
State := eState;
END_GET
END_PROPERTY

/// aktueller Schritt
{attribute 'monitoring':='call'}
PROPERTY Step : INT
GET
Step := nStep;
END_GET
END_PROPERTY

METHOD StepDefinition : BOOL
VAR_INPUT
	clearText				: STRING;
	maxStepTime				: TIME;
END_VAR
sClearText := clearText;
tmaxStepTime := maxStepTime;
END_METHOD

METHOD Stepping
VAR_INPUT
END_VAR
bStepping := TRUE;
END_METHOD

/// Schritt Timeout - flag 
{attribute 'monitoring':='variable'}
PROPERTY TimeoutStep : BOOL
GET
TimeoutStep := bTimeoutStep;
END_GET
END_PROPERTY

PROPERTY Waiting : BOOL
GET
Waiting := eState = eSequenceState_waiting;
END_GET
SET
IF Waiting AND eState = eSequenceState_running THEN
	eState := eSequenceState_waiting;	
ELSIF NOT Waiting AND eState = eSequenceState_waiting THEN
	eState := eSequenceState_running;	
END_IF
END_SET
END_PROPERTY

END_FUNCTION_BLOCK

// ---- Utilities/Composition/FB_CompositionBase.TcPOU
FUNCTION_BLOCK FB_CompositionBase EXTENDS FB_ComponentBase
VAR	
	aComponents					: ARRAY[0..iMaxIdxComponent] OF ITFComponent;
	eCompostitionState			: E_ComponentState;
	nComponent					: INT := -1;	
	nErrComponent				: INT;
	sErrComponentName			: STRING;
END_VAR

///
/// 
/// HF/www.asma.at/02.2018
///

PROPERTY ComponentState : E_ComponentState
GET
ComponentState := eCompostitionState;
END_GET
END_PROPERTY

PROPERTY CompostitionState : E_ComponentState
GET
CompostitionState := eCompostitionState;
END_GET
END_PROPERTY

METHOD GetComponent : POINTER TO FB_ComponentBase
VAR_INPUT
	nSubComp			:INT;	
END_VAR

VAR
	ptTmp				: POINTER TO FB_ComponentBase;
	bFound				: BOOL;
END_VAR
bFound := __QUERYPOINTER(aComponents[nSubComp], ptTmp);

IF bFound THEN
	GetComponent := ptTmp;
ELSE
	GetComponent := 0;
END_IF
END_METHOD

METHOD GetItfComponent : ITFComponent
VAR_INPUT
	nSubComp			:INT;	
END_VAR
GetItfComponent := aComponents[nSubComp];
END_METHOD

METHOD HaltAll
VAR
	iIdx			: INT;
	itfAxis			: ITFMotionComponent;
	//ptLifting		: POINTER TO FB_LiftingUnit;
END_VAR
// run all components
FOR iIdx := 0 TO GVL_CONST.iMaxIdxComponent DO
	// chk valid pointer
	IF aComponents[iIdx] <> 0 THEN
		// chk component is active
		IF NOT aComponents[iIdx].Active THEN
			CONTINUE;
		END_IF
 
		IF __QUERYINTERFACE(aComponents[iIdx], itfAxis) THEN
			itfAxis.Halt();	
		END_IF
		
	END_IF
END_FOR
END_METHOD

METHOD LoadComponents
VAR_INPUT
END_VAR
nComponent := 0;
MEMSET(ADR(aComponents), 0, SIZEOF(aComponents));
eCompostitionState := E_ComponentState.eComponentState_none;
END_METHOD

/// Registrierung von PM Sub-Komponenten.
METHOD RegisterComponent
VAR_INPUT
	ID				: INT := 0;
	fbComponent  	: ITFComponent;
END_VAR
IF fbComponent = 0 THEN
	sClearText := 'invalid sub-component pointer!';
	eCompostitionState := eComponentState_error;
	RETURN;
END_IF

// register sub-component
fbComponent.ID := ID;
fbComponent.SetEventLogReference(fbEventlog);
aComponents[nComponent] := fbComponent;

// increment counter
IF nComponent < GVL_CONST.iMaxIdxComponent THEN
	nComponent := nComponent + 1;
ELSE
	sClearText := 'max. component index overrun!';
	eCompostitionState := eComponentState_error;
	RETURN;
END_IF
END_METHOD

/// Reset component logic
{attribute 'object_name' := 'Reset'}
METHOD Reset
/// abstract base logic reset

sLastError := sEmpty;
MEMSET(ADR(stLastEvent), 0, SIZEOF(ST_EVENT));

// default: set state to ready
eState := E_ComponentState.eComponentState_ready;

/// reset all components				
ResetComponents(FALSE, FALSE, 0, 0);
END_METHOD

METHOD ResetComponents
VAR_INPUT
	bOnlyActive			: BOOL;
	bOnlyNotRunning		: BOOL;
	eComponentType		: E_ComponentType;
	eExpectType			: E_ComponentType;
END_VAR

VAR
	iIdx				: INT;
END_VAR
/// reset all components				
FOR iIdx := 0 TO GVL_CONST.iMaxIdxComponent DO
	IF aComponents[iIdx] <> 0 THEN
		
		IF aComponents[iIdx].State = eComponentState_running AND bOnlyNotRunning THEN
			CONTINUE;
		END_IF
	
		IF bOnlyActive AND NOT aComponents[iIdx].Active THEN
			CONTINUE;
		END_IF
		
		IF (eComponentType = eComponentType_none OR aComponents[iIdx].Typ = eComponentType) AND
		   (eExpectType = eComponentType_none OR aComponents[iIdx].Typ <> eExpectType) THEN
			aComponents[iIdx].Reset();		
		END_IF
		
	END_IF
END_FOR
END_METHOD

/// Run component logic
{attribute 'object_name' := 'Run'}
METHOD Run : E_ComponentState

VAR
	iIdx			: INT;
END_VAR
/// abstract base logic run

// only rdy state may lead to run
IF eState = E_ComponentState.eComponentState_ready THEN
	eState := E_ComponentState.eComponentState_running;
END_IF


// run HMI & logger
//fbEventLog.Run();

// latch resetting state
//bIsResetting := (eState = eComponentState_resetting);

/// run components

// set overall component state, prio:
// 1. E_ComponentState.eComponentState_error		( --> at least one has error)
// 2. E_ComponentState.eComponentState_none			( --> at least one state is not set)
// 3. E_ComponentState.eComponentState_resetting	( --> at least one is rsetting)
// 4. E_ComponentState.eComponentState_ready		( --> at least one is in ready state)
// 5. E_ComponentState.eComponentState_running		( --> all active are running)

// init with running state
eCompostitionState := eComponentState_running;

// run all components
FOR iIdx := 0 TO GVL_CONST.iMaxIdxComponent DO
	// chk valid pointer
	IF aComponents[iIdx] <> 0 THEN
		// chk component is active
		IF aComponents[iIdx].Active THEN
			// run component and get it's state 
			CASE aComponents[iIdx].Run() OF
				eComponentState_error:
					IF nErrComponent = 0 THEN
						nErrComponent := iIdx;
						sErrComponentName := aComponents[iIdx].Name;
					END_IF
					eCompostitionState := eComponentState_error;	
					
				eComponentState_none:
					IF eCompostitionState <> eComponentState_error THEN
						eCompostitionState := eComponentState_none;
					END_IF
					
				eComponentState_resetting:
					IF eCompostitionState <> eComponentState_error AND eCompostitionState <> eComponentState_none THEN
						eCompostitionState := eComponentState_resetting;
					END_IF
					
				eComponentState_ready:
					IF eCompostitionState = eComponentState_running THEN
						eCompostitionState := eComponentState_ready;
					END_IF					
			END_CASE
		END_IF
	END_IF
END_FOR

eState := eCompostitionState;


Run := eState;
END_METHOD

END_FUNCTION_BLOCK

// ---- Utilities/Component/FB_ComponentBase.TcPOU
/// Abstract base FB for components
{attribute 'enable_dynamic_creation' := ''}
{attribute 'reflection' := ''}
FUNCTION_BLOCK FB_ComponentBase IMPLEMENTS ITFComponent
VAR
	/// Unique ID of this instance (cam be used as index: P_ComponentPool.aComponents[iID]...)
	iId				: INT := -1;
	/// component active flag
	bActive			: BOOL;
	/// component state
	eState			: E_ComponentState;
	/// clear text info
	sClearText		: T_MaxString;
	/// last error debug info
	sLastError		: T_MaxString;	
	/// component type
	eTyp			: E_ComponentType;
	/// EventLog reference
	fbEventLog		: REFERENCE TO FB_EventLog;
	/// Last Event
	stLastEvent		: ST_Event;
	ptLastEvent		: POINTER TO ST_Event;
	
	
	/// Bereich
	eMachineArea	: E_MachineArea;
	/// component name
	sName			: STRING;
	/// BMK name
	sBMK			: STRING;
	/// path of this FB (e.g. for log: P_ComponentPool.fbVirtualMaster)
	{attribute 'no_init' := ''}
	{attribute 'instance-path' := ''}
	sPath			: STRING;	

END_VAR

///
/// Abstract base FB for components
/// TP/www.rmth.at/11.2014
///

/// Get's or set's a value indicating whether this component is active or not.
PROPERTY Active : BOOL
GET
Active := bActive;
END_GET
SET
bActive := Active;
sClearText := SEL(bActive, 'INACTIVE!', 'ACTIVE!');
END_SET
END_PROPERTY

PROPERTY BMK : STRING
GET
BMK := sBMK;
END_GET
SET
sBMK := BMK;
END_SET
END_PROPERTY

/// Get's value representing the component state.
PROPERTY ClearText : String
GET
ClearText := sClearText;
END_GET
END_PROPERTY

/// Unique component ID (cam be used as index: P_ComponentPool.aComponents[eID]...)
PROPERTY ID : INT
GET
ID := iId;
END_GET
SET
iID := Id;
END_SET
END_PROPERTY

/// Get's value representing the component state.
PROPERTY LastError : String
GET
LastError := sLastError;
END_GET
END_PROPERTY

PROPERTY MachineArea : E_MachineArea
GET
MachineArea := eMachineArea;
END_GET
SET
eMachineArea := MachineArea;
END_SET
END_PROPERTY

PROPERTY Name : STRING
GET
Name := sName;
END_GET
SET
sName := Name;
END_SET
END_PROPERTY

PROPERTY Path : String
GET
Path := sPath;
END_GET
END_PROPERTY

/// Reset component logic
{attribute 'object_name' := 'Reset'}
METHOD Reset
/// abstract base logic reset

sLastError := sEmpty;
MEMSET(ADR(stLastEvent), 0, SIZEOF(ST_EVENT));

// default: set state to ready
eState := E_ComponentState.eComponentState_ready;
END_METHOD

/// Run component logic
{attribute 'object_name' := 'Run'}
METHOD Run : E_ComponentState
/// abstract base logic run

// only rdy state may lead to run
IF eState = E_ComponentState.eComponentState_ready THEN
	eState := E_ComponentState.eComponentState_running;
END_IF

Run := eState;

IF stLastEvent.ePriority < E_Priority.ePriority_fault AND eState = E_ComponentState.eComponentState_error THEN
	WriteError(E_Event.eEvent_none, 'unbekannter Fehler');
END_IF
END_METHOD

/// Set EventLog reference
METHOD SetEventLogReference
VAR_IN_OUT
	/// HMI access provider.
	fbEventLogRef	: FB_EventLog;
END_VAR
fbEventLog REF= fbEventLogRef;
END_METHOD

/// Get's value representing the component state.
PROPERTY State : E_ComponentState
GET
State := eState;
END_GET
END_PROPERTY

/// Get's value representing the component state.
PROPERTY StateAsString : STRING
GET
CASE eState OF

	eComponentState_none :
		StateAsString := 'undefiniert';
	/// Component is resetting
	eComponentState_resetting:
		StateAsString := 'wird zurückgesetzt';
	/// Component is ready
	eComponentState_ready:
		StateAsString := 'ist bereit';
	/// Component is running
	eComponentState_running:
		StateAsString := 'wird ausgeführt';
	/// Component has error
	eComponentState_error:
		StateAsString := 'ist fehlerhaft';

END_CASE
END_GET
END_PROPERTY

PROPERTY Typ : E_ComponentType
GET
Typ := eTyp;
END_GET
END_PROPERTY

